LIN {X 0,Y 573.004,Z 629.89,A -85,B 0,C 180,E1 -2246.484,E2 -2246.484} C_VEL
LIN {X 0,Y 572.937,Z 632.192,A -85,B 0,C 180,E1 -2247.891,E2 -2247.891} C_VEL
LIN {X 0,Y 572.938,Z 633.349,A -85,B 0,C 180,E1 -2249.297,E2 -2249.297} C_VEL
LIN {X 0,Y 572.938,Z 633.349,A -85,B 0,C 180,E1 -2250.703,E2 -2250.703} C_VEL
LIN {X 0,Y 572.937,Z 632.19,A -85,B 0,C 180,E1 -2252.109,E2 -2252.109} C_VEL
LIN {X 0,Y 573.004,Z 629.886,A -85,B 0,C 180,E1 -2253.516,E2 -2253.516} C_VEL
LIN {X 0,Y 572.951,Z 626.385,A -85,B 0,C 180,E1 -2254.926,E2 -2254.926} C_VEL
LIN {X 0,Y 573.012,Z 621.608,A -85,B 0,C 180,E1 -2256.338,E2 -2256.338} C_VEL
LIN {X 0,Y 573.094,Z 615.422,A -85,B 0,C 180,E1 -2257.753,E2 -2257.753} C_VEL
LIN {X 0,Y 573.136,Z 607.648,A -85,B 0,C 180,E1 -2259.173,E2 -2259.173} C_VEL
LIN {X 0,Y 573.27,Z 599.368,A -85,B 0,C 180,E1 -2260.418,E2 -2260.418} C_VEL
LIN {X 0,Y 573.386,Z 589.391,A -85,B 0,C 180,E1 -2261.668,E2 -2261.668} C_VEL
LIN {X 0,Y 573.568,Z 579.188,A -85,B 0,C 180,E1 -2262.742,E2 -2262.742} C_VEL
LIN {X 0,Y 573.705,Z 567.019,A -85,B 0,C 180,E1 -2263.82,E2 -2263.82} C_VEL
LIN {X 0,Y 573.963,Z 553.905,A -85,B 0,C 180,E1 -2264.781,E2 -2264.781} C_VEL
LIN {X 0,Y 574.144,Z 539.872,A -85,B 0,C 180,E1 -2265.622,E2 -2265.622} C_VEL
LIN {X 0,Y 574.34,Z 525.8,A -85,B 0,C 180,E1 -2266.301,E2 -2266.301} C_VEL
LIN {X 0,Y 574.564,Z 511.306,A -85,B 0,C 180,E1 -2266.842,E2 -2266.842} C_VEL
LIN {X 0,Y 574.707,Z 496.013,A -85,B 0,C 180,E1 -2267.261,E2 -2267.261} C_VEL
LIN {X 0,Y 574.798,Z 480.641,A -85,B 0,C 180,E1 -2267.532,E2 -2267.532} C_VEL
LIN {X 0,Y 575.183,Z 328.245,A -85,B 0,C 180,E1 -2269.486,E2 -2269.486} C_VEL
LIN {X 0,Y 574.002,Z 321.806,A -85,B 0,C 180,E1 -2269.623,E2 -2269.623} C_VEL
LIN {X 0,Y 574.351,Z 296.393,A -85,B 0,C 180,E1 -2272.671,E2 -2272.671} C_VEL
LIN {X 0,Y 574.622,Z 274.45,A -85,B 0,C 180,E1 -2275.345,E2 -2275.345} C_VEL
LIN {X 0,Y 573.935,Z 269.691,A -85,B 0,C 180,E1 -2275.961,E2 -2275.961} C_VEL
LIN {X 0,Y 573.238,Z 266.709,A -85,B 0,C 180,E1 -2276.376,E2 -2276.376} C_VEL
LIN {X 0,Y 573.259,Z 266.699,A -85,B 0,C 180,E1 -2279.366,E2 -2279.366} C_VEL
LIN {X 0,Y 573.246,Z 266.708,A -85,B 0,C 180,E1 -2282.227,E2 -2282.227} C_VEL
LIN {X 0,Y 573.219,Z 266.705,A -85,B 0,C 180,E1 -2284.769,E2 -2284.769} C_VEL
LIN {X 0,Y 573.22,Z 266.708,A -85,B 0,C 180,E1 -2287.808,E2 -2287.808} C_VEL
LIN {X 0,Y 573.244,Z 266.702,A -85,B 0,C 180,E1 -2290.524,E2 -2290.524} C_VEL
LIN {X 0,Y 573.196,Z 266.705,A -85,B 0,C 180,E1 -2293.362,E2 -2293.362} C_VEL
LIN {X 0,Y 573.203,Z 266.709,A -85,B 0,C 180,E1 -2296.335,E2 -2296.335} C_VEL
LIN {X 0,Y 573.201,Z 266.707,A -85,B 0,C 180,E1 -2298.54,E2 -2298.54} C_VEL
LIN {X 0,Y 573.227,Z 266.701,A -85,B 0,C 180,E1 -2301.297,E2 -2301.297} C_VEL
LIN {X 0,Y 573.181,Z 266.715,A -85,B 0,C 180,E1 -2304.022,E2 -2304.022} C_VEL
LIN {X 0,Y 573.225,Z 266.702,A -85,B 0,C 180,E1 -2306.514,E2 -2306.514} C_VEL
LIN {X 0,Y 573.216,Z 266.703,A -85,B 0,C 180,E1 -2309.119,E2 -2309.119} C_VEL
LIN {X 0,Y 573.215,Z 266.71,A -85,B 0,C 180,E1 -2311.976,E2 -2311.976} C_VEL
LIN {X 0,Y 573.2,Z 266.705,A -85,B 0,C 180,E1 -2314.587,E2 -2314.587} C_VEL
LIN {X 0,Y 573.231,Z 266.7,A -85,B 0,C 180,E1 -2316.9,E2 -2316.9} C_VEL
LIN {X 0,Y 573.241,Z 266.701,A -85,B 0,C 180,E1 -2319.172,E2 -2319.172} C_VEL
LIN {X 0,Y 573.194,Z 266.709,A -85,B 0,C 180,E1 -2321.409,E2 -2321.409} C_VEL
LIN {X 0,Y 573.209,Z 266.704,A -85,B 0,C 180,E1 -2324.35,E2 -2324.35} C_VEL
LIN {X 0,Y 573.201,Z 266.701,A -85,B 0,C 180,E1 -2326.528,E2 -2326.528} C_VEL
LIN {X 0,Y 573.218,Z 266.705,A -85,B 0,C 180,E1 -2329.401,E2 -2329.401} C_VEL
LIN {X 0,Y 573.202,Z 266.705,A -85,B 0,C 180,E1 -2332.248,E2 -2332.248} C_VEL
LIN {X 0,Y 573.283,Z 266.695,A -85,B 0,C 180,E1 -2335.076,E2 -2335.076} C_VEL
LIN {X 0,Y 573.279,Z 266.697,A -85,B 0,C 180,E1 -2337.891,E2 -2337.891} C_VEL
LIN {X 0,Y 573.287,Z 266.696,A -85,B 0,C 180,E1 -2339.999,E2 -2339.999} C_VEL
LIN {X 0,Y 573.266,Z 266.696,A -85,B 0,C 180,E1 -2342.81,E2 -2342.81} C_VEL
LIN {X 0,Y 573.257,Z 266.7,A -85,B 0,C 180,E1 -2345.627,E2 -2345.627} C_VEL
LIN {X 0,Y 573.209,Z 266.701,A -85,B 0,C 180,E1 -2348.459,E2 -2348.459} C_VEL
LIN {X 0,Y 573.26,Z 266.705,A -85,B 0,C 180,E1 -2351.311,E2 -2351.311} C_VEL
LIN {X 0,Y 573.213,Z 266.701,A -85,B 0,C 180,E1 -2354.401,E2 -2354.401} C_VEL
LIN {X 0,Y 573.224,Z 266.703,A -85,B 0,C 180,E1 -2357.111,E2 -2357.111} C_VEL
LIN {X 0,Y 573.214,Z 266.702,A -85,B 0,C 180,E1 -2360.076,E2 -2360.076} C_VEL
LIN {X 0,Y 573.204,Z 266.703,A -85,B 0,C 180,E1 -2362.337,E2 -2362.337} C_VEL
LIN {X 0,Y 573.18,Z 266.706,A -85,B 0,C 180,E1 -2364.332,E2 -2364.332} C_VEL
LIN {X 0,Y 572.541,Z 266.791,A -85,B 0,C 180,E1 -2364.919,E2 -2364.919} C_VEL
LIN {X 0,Y 569.711,Z 267.148,A -85,B 0,C 180,E1 -2365.87,E2 -2365.87} C_VEL
LIN {X 0,Y 567.294,Z 267.45,A -85,B 0,C 180,E1 -2366.636,E2 -2366.636} C_VEL
LIN {X 0,Y 566.238,Z 267.577,A -85,B 0,C 180,E1 -2367.227,E2 -2367.227} C_VEL
LIN {X 0,Y 566.143,Z 267.586,A -85,B 0,C 180,E1 -2367.428,E2 -2367.428} C_VEL
LIN {X 0,Y 566.147,Z 267.584,A -85,B 0,C 180,E1 -2369.77,E2 -2369.77} C_VEL
LIN {X 0,Y 566.183,Z 267.579,A -85,B 0,C 180,E1 -2372.428,E2 -2372.428} C_VEL
LIN {X 0,Y 566.151,Z 267.588,A -85,B 0,C 180,E1 -2374.987,E2 -2374.987} C_VEL
LIN {X 0,Y 566.174,Z 267.582,A -85,B 0,C 180,E1 -2377.46,E2 -2377.46} C_VEL
LIN {X 0,Y 566.19,Z 267.577,A -85,B 0,C 180,E1 -2380.198,E2 -2380.198} C_VEL
LIN {X 0,Y 566.176,Z 267.588,A -85,B 0,C 180,E1 -2383.054,E2 -2383.054} C_VEL
LIN {X 0,Y 566.141,Z 267.581,A -85,B 0,C 180,E1 -2386.052,E2 -2386.052} C_VEL
LIN {X 0,Y 566.153,Z 267.59,A -85,B 0,C 180,E1 -2388.859,E2 -2388.859} C_VEL
LIN {X 0,Y 566.189,Z 267.579,A -85,B 0,C 180,E1 -2391.441,E2 -2391.441} C_VEL
LIN {X 0,Y 566.155,Z 267.582,A -85,B 0,C 180,E1 -2394.308,E2 -2394.308} C_VEL
LIN {X 0,Y 566.185,Z 267.588,A -85,B 0,C 180,E1 -2396.896,E2 -2396.896} C_VEL
LIN {X 0,Y 566.158,Z 267.582,A -85,B 0,C 180,E1 -2399.406,E2 -2399.406} C_VEL
LIN {X 0,Y 566.193,Z 267.577,A -85,B 0,C 180,E1 -2401.857,E2 -2401.857} C_VEL
LIN {X 0,Y 566.189,Z 267.579,A -85,B 0,C 180,E1 -2404.25,E2 -2404.25} C_VEL
LIN {X 0,Y 566.152,Z 267.59,A -85,B 0,C 180,E1 -2406.718,E2 -2406.718} C_VEL
LIN {X 0,Y 566.193,Z 267.576,A -85,B 0,C 180,E1 -2409.662,E2 -2409.662} C_VEL
LIN {X 0,Y 566.179,Z 267.588,A -85,B 0,C 180,E1 -2412.668,E2 -2412.668} C_VEL
LIN {X 0,Y 566.208,Z 267.575,A -85,B 0,C 180,E1 -2415.626,E2 -2415.626} C_VEL
LIN {X 0,Y 566.259,Z 267.579,A -85,B 0,C 180,E1 -2418.652,E2 -2418.652} C_VEL
LIN {X 0,Y 566.187,Z 267.578,A -85,B 0,C 180,E1 -2421.434,E2 -2421.434} C_VEL
LIN {X 0,Y 566.242,Z 267.576,A -85,B 0,C 180,E1 -2424.301,E2 -2424.301} C_VEL
LIN {X 0,Y 566.252,Z 267.572,A -85,B 0,C 180,E1 -2427.866,E2 -2427.866} C_VEL
LIN {X 0,Y 566.294,Z 267.574,A -85,B 0,C 180,E1 -2430.711,E2 -2430.711} C_VEL
LIN {X 0,Y 566.167,Z 267.583,A -85,B 0,C 180,E1 -2433.558,E2 -2433.558} C_VEL
LIN {X 0,Y 566.237,Z 267.575,A -85,B 0,C 180,E1 -2435.698,E2 -2435.698} C_VEL
LIN {X 0,Y 566.214,Z 267.629,A -85,B 0,C 180,E1 -2436.562,E2 -2436.562} C_VEL
LIN {X 0,Y 567.18,Z 272.823,A -85,B 0,C 180,E1 -2437.357,E2 -2437.357} C_VEL
LIN {X 0,Y 566.994,Z 288.919,A -85,B 0,C 180,E1 -2439.632,E2 -2439.632} C_VEL
LIN {X 0,Y 566.937,Z 293.131,A -85,B 0,C 180,E1 -2440.197,E2 -2440.197} C_VEL
LIN {X 0,Y 568.464,Z 300.492,A -85,B 0,C 180,E1 -2440.349,E2 -2440.349} C_VEL
LIN {X 0,Y 568.012,Z 456.718,A -85,B 0,C 180,E1 -2442.391,E2 -2442.391} C_VEL
LIN {X 0,Y 567.847,Z 471.71,A -85,B 0,C 180,E1 -2442.712,E2 -2442.712} C_VEL
LIN {X 0,Y 567.619,Z 487.068,A -85,B 0,C 180,E1 -2443.196,E2 -2443.196} C_VEL
LIN {X 0,Y 567.401,Z 501.304,A -85,B 0,C 180,E1 -2443.794,E2 -2443.794} C_VEL
LIN {X 0,Y 567.186,Z 515.574,A -85,B 0,C 180,E1 -2444.555,E2 -2444.555} C_VEL
LIN {X 0,Y 566.934,Z 529.252,A -85,B 0,C 180,E1 -2445.457,E2 -2445.457} C_VEL
LIN {X 0,Y 566.673,Z 542.03,A -85,B 0,C 180,E1 -2446.481,E2 -2446.481} C_VEL
LIN {X 0,Y 566.461,Z 552.788,A -85,B 0,C 180,E1 -2447.509,E2 -2447.509} C_VEL
LIN {X 0,Y 566.31,Z 562.764,A -85,B 0,C 180,E1 -2448.636,E2 -2448.636} C_VEL
LIN {X 0,Y 566.164,Z 572.566,A -85,B 0,C 180,E1 -2449.959,E2 -2449.959} C_VEL
LIN {X 0,Y 566.028,Z 581.205,A -85,B 0,C 180,E1 -2451.379,E2 -2451.379} C_VEL
LIN {X 0,Y 565.992,Z 587.484,A -85,B 0,C 180,E1 -2452.639,E2 -2452.639} C_VEL
LIN {X 0,Y 565.929,Z 593.647,A -85,B 0,C 180,E1 -2454.192,E2 -2454.192} C_VEL
LIN {X 0,Y 565.877,Z 598.273,A -85,B 0,C 180,E1 -2455.764,E2 -2455.764} C_VEL
LIN {X 0,Y 565.824,Z 601.432,A -85,B 0,C 180,E1 -2457.358,E2 -2457.358} C_VEL
LIN {X 0,Y 565.831,Z 603.143,A -85,B 0,C 180,E1 -2458.973,E2 -2458.973} C_VEL
LIN {X 0,Y 565.866,Z 603.382,A -85,B 0,C 180,E1 -2460.61,E2 -2460.61} C_VEL
LIN {X 0,Y 565.841,Z 602.082,A -85,B 0,C 180,E1 -2462.28,E2 -2462.28} C_VEL
LIN {X 0,Y 565.867,Z 599.727,A -85,B 0,C 180,E1 -2463.685,E2 -2463.685} C_VEL
LIN {X 0,Y 565.899,Z 595.585,A -85,B 0,C 180,E1 -2465.303,E2 -2465.303} C_VEL
LIN {X 0,Y 565.943,Z 591.112,A -85,B 0,C 180,E1 -2466.588,E2 -2466.588} C_VEL
LIN {X 0,Y 566,Z 585.273,A -85,B 0,C 180,E1 -2467.924,E2 -2467.924} C_VEL
LIN {X 0,Y 566.09,Z 577.948,A -85,B 0,C 180,E1 -2469.283,E2 -2469.283} C_VEL
LIN {X 0,Y 566.222,Z 568.957,A -85,B 0,C 180,E1 -2470.648,E2 -2470.648} C_VEL
LIN {X 0,Y 566.322,Z 559.209,A -85,B 0,C 180,E1 -2471.879,E2 -2471.879} C_VEL
LIN {X 0,Y 566.544,Z 548.415,A -85,B 0,C 180,E1 -2473.02,E2 -2473.02} C_VEL
LIN {X 0,Y 566.795,Z 536.367,A -85,B 0,C 180,E1 -2474.087,E2 -2474.087} C_VEL
LIN {X 0,Y 567.041,Z 523.201,A -85,B 0,C 180,E1 -2475.055,E2 -2475.055} C_VEL
LIN {X 0,Y 567.272,Z 509.632,A -85,B 0,C 180,E1 -2475.873,E2 -2475.873} C_VEL
LIN {X 0,Y 567.52,Z 495.08,A -85,B 0,C 180,E1 -2476.575,E2 -2476.575} C_VEL
LIN {X 0,Y 567.733,Z 479.651,A -85,B 0,C 180,E1 -2477.147,E2 -2477.147} C_VEL
LIN {X 0,Y 567.942,Z 464.183,A -85,B 0,C 180,E1 -2477.557,E2 -2477.557} C_VEL
LIN {X 0,Y 568.026,Z 447.504,A -85,B 0,C 180,E1 -2477.834,E2 -2477.834} C_VEL
LIN {X 0,Y 568.365,Z 299.674,A -85,B 0,C 180,E1 -2479.755,E2 -2479.755} C_VEL
LIN {X 0,Y 566.896,Z 292.8,A -85,B 0,C 180,E1 -2479.917,E2 -2479.917} C_VEL
LIN {X 0,Y 567.195,Z 273.626,A -85,B 0,C 180,E1 -2482.619,E2 -2482.619} C_VEL
LIN {X 0,Y 566.221,Z 267.583,A -85,B 0,C 180,E1 -2483.562,E2 -2483.562} C_VEL
LIN {X 0,Y 566.211,Z 267.578,A -85,B 0,C 180,E1 -2486.264,E2 -2486.264} C_VEL
LIN {X 0,Y 566.187,Z 267.581,A -85,B 0,C 180,E1 -2488.922,E2 -2488.922} C_VEL
LIN {X 0,Y 566.182,Z 267.584,A -85,B 0,C 180,E1 -2491.048,E2 -2491.048} C_VEL
LIN {X 0,Y 566.231,Z 267.582,A -85,B 0,C 180,E1 -2493.461,E2 -2493.461} C_VEL
LIN {X 0,Y 566.182,Z 267.583,A -85,B 0,C 180,E1 -2495.82,E2 -2495.82} C_VEL
LIN {X 0,Y 566.201,Z 267.58,A -85,B 0,C 180,E1 -2498.904,E2 -2498.904} C_VEL
LIN {X 0,Y 566.198,Z 267.585,A -85,B 0,C 180,E1 -2501.174,E2 -2501.174} C_VEL
LIN {X 0,Y 566.204,Z 267.583,A -85,B 0,C 180,E1 -2503.414,E2 -2503.414} C_VEL
LIN {X 0,Y 566.186,Z 267.579,A -85,B 0,C 180,E1 -2506.36,E2 -2506.36} C_VEL
LIN {X 0,Y 566.219,Z 267.577,A -85,B 0,C 180,E1 -2508.676,E2 -2508.676} C_VEL
LIN {X 0,Y 566.192,Z 267.582,A -85,B 0,C 180,E1 -2511.435,E2 -2511.435} C_VEL
LIN {X 0,Y 566.246,Z 267.571,A -85,B 0,C 180,E1 -2514.303,E2 -2514.303} C_VEL
LIN {X 0,Y 566.257,Z 267.57,A -85,B 0,C 180,E1 -2517.867,E2 -2517.867} C_VEL
LIN {X 0,Y 566.298,Z 267.571,A -85,B 0,C 180,E1 -2520.712,E2 -2520.712} C_VEL
LIN {X 0,Y 566.264,Z 267.577,A -85,B 0,C 180,E1 -2522.847,E2 -2522.847} C_VEL
LIN {X 0,Y 566.232,Z 267.573,A -85,B 0,C 180,E1 -2525.7,E2 -2525.7} C_VEL
LIN {X 0,Y 566.191,Z 267.577,A -85,B 0,C 180,E1 -2527.849,E2 -2527.849} C_VEL
LIN {X 0,Y 566.225,Z 267.582,A -85,B 0,C 180,E1 -2530.731,E2 -2530.731} C_VEL
LIN {X 0,Y 566.173,Z 267.579,A -85,B 0,C 180,E1 -2533.643,E2 -2533.643} C_VEL
LIN {X 0,Y 566.201,Z 267.585,A -85,B 0,C 180,E1 -2536.589,E2 -2536.589} C_VEL
LIN {X 0,Y 566.19,Z 267.577,A -85,B 0,C 180,E1 -2539.582,E2 -2539.582} C_VEL
LIN {X 0,Y 566.178,Z 267.58,A -85,B 0,C 180,E1 -2541.864,E2 -2541.864} C_VEL
LIN {X 0,Y 566.168,Z 267.582,A -85,B 0,C 180,E1 -2545.022,E2 -2545.022} C_VEL
LIN {X 0,Y 566.153,Z 267.582,A -85,B 0,C 180,E1 -2547.343,E2 -2547.343} C_VEL
LIN {X 0,Y 566.156,Z 267.583,A -85,B 0,C 180,E1 -2549.772,E2 -2549.772} C_VEL
LIN {X 0,Y 566.184,Z 267.587,A -85,B 0,C 180,E1 -2552.429,E2 -2552.429} C_VEL
LIN {X 0,Y 566.15,Z 267.583,A -85,B 0,C 180,E1 -2554.987,E2 -2554.987} C_VEL
LIN {X 0,Y 566.175,Z 267.58,A -85,B 0,C 180,E1 -2557.463,E2 -2557.463} C_VEL
LIN {X 0,Y 566.171,Z 267.59,A -85,B 0,C 180,E1 -2560.203,E2 -2560.203} C_VEL
LIN {X 0,Y 566.172,Z 267.58,A -85,B 0,C 180,E1 -2563.058,E2 -2563.058} C_VEL
LIN {X 0,Y 566.149,Z 267.592,A -85,B 0,C 180,E1 -2566.055,E2 -2566.055} C_VEL
LIN {X 0,Y 566.168,Z 267.581,A -85,B 0,C 180,E1 -2569.219,E2 -2569.219} C_VEL
LIN {X 0,Y 566.171,Z 267.585,A -85,B 0,C 180,E1 -2571.637,E2 -2571.637} C_VEL
LIN {X 0,Y 566.136,Z 267.589,A -85,B 0,C 180,E1 -2574.307,E2 -2574.307} C_VEL
LIN {X 0,Y 566.205,Z 267.577,A -85,B 0,C 180,E1 -2576.898,E2 -2576.898} C_VEL
LIN {X 0,Y 566.174,Z 267.584,A -85,B 0,C 180,E1 -2579.408,E2 -2579.408} C_VEL
LIN {X 0,Y 566.185,Z 267.587,A -85,B 0,C 180,E1 -2581.857,E2 -2581.857} C_VEL
LIN {X 0,Y 566.163,Z 267.606,A -85,B 0,C 180,E1 -2583.425,E2 -2583.425} C_VEL
LIN {X 0,Y 567.69,Z 274.251,A -85,B 0,C 180,E1 -2584.324,E2 -2584.324} C_VEL
LIN {X 0,Y 567.568,Z 291.068,A -85,B 0,C 180,E1 -2586.394,E2 -2586.394} C_VEL
LIN {X 0,Y 567.283,Z 312.004,A -85,B 0,C 180,E1 -2588.945,E2 -2588.945} C_VEL
LIN {X 0,Y 567.116,Z 321.972,A -85,B 0,C 180,E1 -2590.143,E2 -2590.143} C_VEL
LIN {X 0,Y 568.492,Z 329.339,A -85,B 0,C 180,E1 -2590.29,E2 -2590.29} C_VEL
LIN {X 0,Y 567.986,Z 487.947,A -85,B 0,C 180,E1 -2592.364,E2 -2592.364} C_VEL
LIN {X 0,Y 567.854,Z 503.728,A -85,B 0,C 180,E1 -2592.721,E2 -2592.721} C_VEL
LIN {X 0,Y 567.607,Z 519.055,A -85,B 0,C 180,E1 -2593.223,E2 -2593.223} C_VEL
LIN {X 0,Y 567.445,Z 532.788,A -85,B 0,C 180,E1 -2593.82,E2 -2593.82} C_VEL
LIN {X 0,Y 567.151,Z 546.258,A -85,B 0,C 180,E1 -2594.549,E2 -2594.549} C_VEL
LIN {X 0,Y 566.931,Z 558.534,A -85,B 0,C 180,E1 -2595.36,E2 -2595.36} C_VEL
LIN {X 0,Y 566.672,Z 571.298,A -85,B 0,C 180,E1 -2596.371,E2 -2596.371} C_VEL
LIN {X 0,Y 566.491,Z 582.755,A -85,B 0,C 180,E1 -2597.461,E2 -2597.461} C_VEL
LIN {X 0,Y 566.269,Z 593.317,A -85,B 0,C 180,E1 -2598.659,E2 -2598.659} C_VEL
LIN {X 0,Y 566.208,Z 601.86,A -85,B 0,C 180,E1 -2599.813,E2 -2599.813} C_VEL
LIN {X 0,Y 566.057,Z 609.737,A -85,B 0,C 180,E1 -2601.072,E2 -2601.072} C_VEL
LIN {X 0,Y 565.998,Z 617.092,A -85,B 0,C 180,E1 -2602.509,E2 -2602.509} C_VEL
LIN {X 0,Y 565.956,Z 622.924,A -85,B 0,C 180,E1 -2603.941,E2 -2603.941} C_VEL
LIN {X 0,Y 565.866,Z 626.387,A -85,B 0,C 180,E1 -2605.013,E2 -2605.013} C_VEL
LIN {X 0,Y 565.909,Z 629.89,A -85,B 0,C 180,E1 -2606.44,E2 -2606.44} C_VEL
LIN {X 0,Y 565.838,Z 632.192,A -85,B 0,C 180,E1 -2607.865,E2 -2607.865} C_VEL
LIN {X 0,Y 565.838,Z 633.349,A -85,B 0,C 180,E1 -2609.289,E2 -2609.289} C_VEL
LIN {X 0,Y 565.838,Z 633.348,A -85,B 0,C 180,E1 -2610.712,E2 -2610.712} C_VEL
LIN {X 0,Y 565.838,Z 632.189,A -85,B 0,C 180,E1 -2612.136,E2 -2612.136} C_VEL
LIN {X 0,Y 565.909,Z 629.886,A -85,B 0,C 180,E1 -2613.56,E2 -2613.56} C_VEL
LIN {X 0,Y 565.867,Z 626.385,A -85,B 0,C 180,E1 -2614.988,E2 -2614.988} C_VEL
LIN {X 0,Y 565.956,Z 622.924,A -85,B 0,C 180,E1 -2616.059,E2 -2616.059} C_VEL
LIN {X 0,Y 565.998,Z 617.087,A -85,B 0,C 180,E1 -2617.492,E2 -2617.492} C_VEL
LIN {X 0,Y 566.058,Z 609.73,A -85,B 0,C 180,E1 -2618.928,E2 -2618.928} C_VEL
LIN {X 0,Y 566.209,Z 601.855,A -85,B 0,C 180,E1 -2620.188,E2 -2620.188} C_VEL
LIN {X 0,Y 566.31,Z 592.39,A -85,B 0,C 180,E1 -2621.453,E2 -2621.453} C_VEL
LIN {X 0,Y 566.492,Z 582.748,A -85,B 0,C 180,E1 -2622.539,E2 -2622.539} C_VEL
LIN {X 0,Y 566.672,Z 571.295,A -85,B 0,C 180,E1 -2623.629,E2 -2623.629} C_VEL
LIN {X 0,Y 566.929,Z 558.68,A -85,B 0,C 180,E1 -2624.63,E2 -2624.63} C_VEL
LIN {X 0,Y 567.153,Z 546.247,A -85,B 0,C 180,E1 -2625.451,E2 -2625.451} C_VEL
LIN {X 0,Y 567.448,Z 532.77,A -85,B 0,C 180,E1 -2626.181,E2 -2626.181} C_VEL
LIN {X 0,Y 567.612,Z 519.047,A -85,B 0,C 180,E1 -2626.777,E2 -2626.777} C_VEL
LIN {X 0,Y 567.848,Z 503.72,A -85,B 0,C 180,E1 -2627.28,E2 -2627.28} C_VEL
LIN {X 0,Y 567.982,Z 488.303,A -85,B 0,C 180,E1 -2627.63,E2 -2627.63} C_VEL
LIN {X 0,Y 568.496,Z 329.245,A -85,B 0,C 180,E1 -2629.711,E2 -2629.711} C_VEL
LIN {X 0,Y 567.138,Z 321.835,A -85,B 0,C 180,E1 -2629.867,E2 -2629.867} C_VEL
LIN {X 0,Y 567.555,Z 294.798,A -85,B 0,C 180,E1 -2633.151,E2 -2633.151} C_VEL
LIN {X 0,Y 567.801,Z 276.029,A -85,B 0,C 180,E1 -2635.453,E2 -2635.453} C_VEL
LIN {X 0,Y 567.026,Z 271.09,A -85,B 0,C 180,E1 -2636.104,E2 -2636.104} C_VEL
LIN {X 0,Y 566.151,Z 267.591,A -85,B 0,C 180,E1 -2636.598,E2 -2636.598} C_VEL
LIN {X 0,Y 566.181,Z 267.582,A -85,B 0,C 180,E1 -2638.954,E2 -2638.954} C_VEL
LIN {X 0,Y 566.189,Z 267.579,A -85,B 0,C 180,E1 -2641.422,E2 -2641.422} C_VEL
LIN {X 0,Y 566.194,Z 267.585,A -85,B 0,C 180,E1 -2643.957,E2 -2643.957} C_VEL
LIN {X 0,Y 566.173,Z 267.584,A -85,B 0,C 180,E1 -2646.571,E2 -2646.571} C_VEL
LIN {X 0,Y 566.209,Z 267.58,A -85,B 0,C 180,E1 -2649.685,E2 -2649.685} C_VEL
LIN {X 0,Y 566.18,Z 267.578,A -85,B 0,C 180,E1 -2652.914,E2 -2652.914} C_VEL
LIN {X 0,Y 566.154,Z 267.59,A -85,B 0,C 180,E1 -2656.053,E2 -2656.053} C_VEL
LIN {X 0,Y 566.154,Z 267.583,A -85,B 0,C 180,E1 -2658.858,E2 -2658.858} C_VEL
LIN {X 0,Y 566.198,Z 267.578,A -85,B 0,C 180,E1 -2661.442,E2 -2661.442} C_VEL
LIN {X 0,Y 566.136,Z 267.587,A -85,B 0,C 180,E1 -2664.305,E2 -2664.305} C_VEL
LIN {X 0,Y 566.194,Z 267.576,A -85,B 0,C 180,E1 -2666.895,E2 -2666.895} C_VEL
LIN {X 0,Y 566.165,Z 267.583,A -85,B 0,C 180,E1 -2669.406,E2 -2669.406} C_VEL
LIN {X 0,Y 566.183,Z 267.588,A -85,B 0,C 180,E1 -2671.855,E2 -2671.855} C_VEL
LIN {X 0,Y 566.17,Z 267.584,A -85,B 0,C 180,E1 -2674.248,E2 -2674.248} C_VEL
LIN {X 0,Y 566.16,Z 267.581,A -85,B 0,C 180,E1 -2676.719,E2 -2676.719} C_VEL
LIN {X 0,Y 566.196,Z 267.586,A -85,B 0,C 180,E1 -2679.661,E2 -2679.661} C_VEL
LIN {X 0,Y 566.161,Z 267.589,A -85,B 0,C 180,E1 -2681.92,E2 -2681.92} C_VEL
LIN {X 0,Y 566.182,Z 267.578,A -85,B 0,C 180,E1 -2684.889,E2 -2684.889} C_VEL
LIN {X 0,Y 566.171,Z 267.584,A -85,B 0,C 180,E1 -2687.817,E2 -2687.817} C_VEL
LIN {X 0,Y 566.131,Z 267.589,A -85,B 0,C 180,E1 -2689.99,E2 -2689.99} C_VEL
LIN {X 0,Y 566.173,Z 267.582,A -85,B 0,C 180,E1 -2692.151,E2 -2692.151} C_VEL
LIN {X 0,Y 566.255,Z 267.569,A -85,B 0,C 180,E1 -2695.015,E2 -2695.015} C_VEL
LIN {X 0,Y 566.252,Z 267.572,A -85,B 0,C 180,E1 -2697.865,E2 -2697.865} C_VEL
LIN {X 0,Y 566.258,Z 267.572,A -85,B 0,C 180,E1 -2699.999,E2 -2699.999} C_VEL
LIN {X 0,Y 566.236,Z 267.572,A -85,B 0,C 180,E1 -2702.845,E2 -2702.845} C_VEL
LIN {X 0,Y 566.222,Z 267.574,A -85,B 0,C 180,E1 -2705.697,E2 -2705.697} C_VEL
LIN {X 0,Y 566.164,Z 267.578,A -85,B 0,C 180,E1 -2708.565,E2 -2708.565} C_VEL
LIN {X 0,Y 566.226,Z 267.582,A -85,B 0,C 180,E1 -2711.453,E2 -2711.453} C_VEL
LIN {X 0,Y 566.163,Z 267.579,A -85,B 0,C 180,E1 -2714.482,E2 -2714.482} C_VEL
LIN {X 0,Y 566.169,Z 267.584,A -85,B 0,C 180,E1 -2717.331,E2 -2717.331} C_VEL
LIN {X 0,Y 566.184,Z 267.583,A -85,B 0,C 180,E1 -2719.58,E2 -2719.58} C_VEL
LIN {X 0,Y 566.17,Z 267.582,A -85,B 0,C 180,E1 -2721.862,E2 -2721.862} C_VEL
LIN {X 0,Y 566.164,Z 267.585,A -85,B 0,C 180,E1 -2725.02,E2 -2725.02} C_VEL
LIN {X 0,Y 566.143,Z 267.586,A -85,B 0,C 180,E1 -2727.428,E2 -2727.428} C_VEL
LIN {X 0,Y 565.453,Z 267.668,A -85,B 0,C 180,E1 -2728.021,E2 -2728.021} C_VEL
LIN {X 0,Y 562.596,Z 268.027,A -85,B 0,C 180,E1 -2728.985,E2 -2728.985} C_VEL
LIN {X 0,Y 560.204,Z 268.324,A -85,B 0,C 180,E1 -2729.761,E2 -2729.761} C_VEL
LIN {X 0,Y 559.188,Z 268.449,A -85,B 0,C 180,E1 -2730.36,E2 -2730.36} C_VEL
LIN {X 0,Y 559.11,Z 268.46,A -85,B 0,C 180,E1 -2730.563,E2 -2730.563} C_VEL
LIN {X 0,Y 559.134,Z 268.459,A -85,B 0,C 180,E1 -2732.715,E2 -2732.715} C_VEL
LIN {X 0,Y 559.101,Z 268.463,A -85,B 0,C 180,E1 -2735.324,E2 -2735.324} C_VEL
LIN {X 0,Y 559.112,Z 268.457,A -85,B 0,C 180,E1 -2738.017,E2 -2738.017} C_VEL
LIN {X 0,Y 559.136,Z 268.461,A -85,B 0,C 180,E1 -2740.812,E2 -2740.812} C_VEL
LIN {X 0,Y 559.118,Z 268.457,A -85,B 0,C 180,E1 -2743.733,E2 -2743.733} C_VEL
LIN {X 0,Y 559.113,Z 268.462,A -85,B 0,C 180,E1 -2746.804,E2 -2746.804} C_VEL
LIN {X 0,Y 559.136,Z 268.463,A -85,B 0,C 180,E1 -2749.187,E2 -2749.187} C_VEL
LIN {X 0,Y 559.112,Z 268.457,A -85,B 0,C 180,E1 -2751.981,E2 -2751.981} C_VEL
LIN {X 0,Y 559.123,Z 268.463,A -85,B 0,C 180,E1 -2754.785,E2 -2754.785} C_VEL
LIN {X 0,Y 559.135,Z 268.459,A -85,B 0,C 180,E1 -2757.364,E2 -2757.364} C_VEL
LIN {X 0,Y 559.125,Z 268.456,A -85,B 0,C 180,E1 -2760.143,E2 -2760.143} C_VEL
LIN {X 0,Y 559.151,Z 268.458,A -85,B 0,C 180,E1 -2763.172,E2 -2763.172} C_VEL
LIN {X 0,Y 559.135,Z 268.457,A -85,B 0,C 180,E1 -2765.494,E2 -2765.494} C_VEL
LIN {X 0,Y 559.151,Z 268.462,A -85,B 0,C 180,E1 -2768.623,E2 -2768.623} C_VEL
LIN {X 0,Y 559.148,Z 268.463,A -85,B 0,C 180,E1 -2770.926,E2 -2770.926} C_VEL
LIN {X 0,Y 559.145,Z 268.454,A -85,B 0,C 180,E1 -2773.947,E2 -2773.947} C_VEL
LIN {X 0,Y 559.149,Z 268.457,A -85,B 0,C 180,E1 -2776.184,E2 -2776.184} C_VEL
LIN {X 0,Y 559.22,Z 268.448,A -85,B 0,C 180,E1 -2779.134,E2 -2779.134} C_VEL
LIN {X 0,Y 559.181,Z 268.452,A -85,B 0,C 180,E1 -2782.053,E2 -2782.053} C_VEL
LIN {X 0,Y 559.236,Z 268.449,A -85,B 0,C 180,E1 -2784.953,E2 -2784.953} C_VEL
LIN {X 0,Y 559.224,Z 268.447,A -85,B 0,C 180,E1 -2787.839,E2 -2787.839} C_VEL
LIN {X 0,Y 559.263,Z 268.451,A -85,B 0,C 180,E1 -2790.72,E2 -2790.72} C_VEL
LIN {X 0,Y 559.229,Z 268.452,A -85,B 0,C 180,E1 -2792.881,E2 -2792.881} C_VEL
LIN {X 0,Y 559.206,Z 268.452,A -85,B 0,C 180,E1 -2795.77,E2 -2795.77} C_VEL
LIN {X 0,Y 559.167,Z 268.531,A -85,B 0,C 180,E1 -2796.359,E2 -2796.359} C_VEL
LIN {X 0,Y 560.336,Z 275.249,A -85,B 0,C 180,E1 -2797.397,E2 -2797.397} C_VEL
LIN {X 0,Y 559.973,Z 292.95,A -85,B 0,C 180,E1 -2799.937,E2 -2799.937} C_VEL
LIN {X 0,Y 561.717,Z 301.086,A -85,B 0,C 180,E1 -2800.11,E2 -2800.11} C_VEL
LIN {X 0,Y 561.232,Z 457.24,A -85,B 0,C 180,E1 -2802.18,E2 -2802.18} C_VEL
LIN {X 0,Y 561.053,Z 472.26,A -85,B 0,C 180,E1 -2802.512,E2 -2802.512} C_VEL
LIN {X 0,Y 560.826,Z 487.052,A -85,B 0,C 180,E1 -2802.985,E2 -2802.985} C_VEL
LIN {X 0,Y 560.56,Z 501.413,A -85,B 0,C 180,E1 -2803.596,E2 -2803.596} C_VEL
LIN {X 0,Y 560.307,Z 515.278,A -85,B 0,C 180,E1 -2804.342,E2 -2804.342} C_VEL
LIN {X 0,Y 560.02,Z 528.256,A -85,B 0,C 180,E1 -2805.199,E2 -2805.199} C_VEL
LIN {X 0,Y 559.735,Z 541.049,A -85,B 0,C 180,E1 -2806.222,E2 -2806.222} C_VEL
LIN {X 0,Y 559.474,Z 553.109,A -85,B 0,C 180,E1 -2807.384,E2 -2807.384} C_VEL
LIN {X 0,Y 559.294,Z 562.821,A -85,B 0,C 180,E1 -2808.498,E2 -2808.498} C_VEL
LIN {X 0,Y 559.109,Z 572.616,A -85,B 0,C 180,E1 -2809.839,E2 -2809.839} C_VEL
LIN {X 0,Y 558.972,Z 580.774,A -85,B 0,C 180,E1 -2811.19,E2 -2811.19} C_VEL
LIN {X 0,Y 558.901,Z 587.518,A -85,B 0,C 180,E1 -2812.552,E2 -2812.552} C_VEL
LIN {X 0,Y 558.851,Z 593.664,A -85,B 0,C 180,E1 -2814.123,E2 -2814.123} C_VEL
LIN {X 0,Y 558.832,Z 597.299,A -85,B 0,C 180,E1 -2815.314,E2 -2815.314} C_VEL
LIN {X 0,Y 558.732,Z 600.82,A -85,B 0,C 180,E1 -2816.924,E2 -2816.924} C_VEL
LIN {X 0,Y 558.72,Z 602.878,A -85,B 0,C 180,E1 -2818.553,E2 -2818.553} C_VEL
LIN {X 0,Y 558.767,Z 603.472,A -85,B 0,C 180,E1 -2820.205,E2 -2820.205} C_VEL
LIN {X 0,Y 558.748,Z 603.093,A -85,B 0,C 180,E1 -2821.21,E2 -2821.21} C_VEL
LIN {X 0,Y 558.745,Z 601.473,A -85,B 0,C 180,E1 -2822.741,E2 -2822.741} C_VEL
LIN {X 0,Y 558.771,Z 599.408,A -85,B 0,C 180,E1 -2823.893,E2 -2823.893} C_VEL
LIN {X 0,Y 558.805,Z 595.656,A -85,B 0,C 180,E1 -2825.346,E2 -2825.346} C_VEL
LIN {X 0,Y 558.866,Z 590.842,A -85,B 0,C 180,E1 -2826.741,E2 -2826.741} C_VEL
LIN {X 0,Y 558.924,Z 585.23,A -85,B 0,C 180,E1 -2828.033,E2 -2828.033} C_VEL
LIN {X 0,Y 559.048,Z 577.898,A -85,B 0,C 180,E1 -2829.408,E2 -2829.408} C_VEL
LIN {X 0,Y 559.195,Z 568.773,A -85,B 0,C 180,E1 -2830.807,E2 -2830.807} C_VEL
LIN {X 0,Y 559.311,Z 559.799,A -85,B 0,C 180,E1 -2831.96,E2 -2831.96} C_VEL
LIN {X 0,Y 559.561,Z 548.98,A -85,B 0,C 180,E1 -2833.13,E2 -2833.13} C_VEL
LIN {X 0,Y 559.85,Z 536.608,A -85,B 0,C 180,E1 -2834.244,E2 -2834.244} C_VEL
LIN {X 0,Y 560.133,Z 523.59,A -85,B 0,C 180,E1 -2835.217,E2 -2835.217} C_VEL
LIN {X 0,Y 560.41,Z 509.502,A -85,B 0,C 180,E1 -2836.079,E2 -2836.079} C_VEL
LIN {X 0,Y 560.677,Z 495.448,A -85,B 0,C 180,E1 -2836.766,E2 -2836.766} C_VEL
LIN {X 0,Y 560.922,Z 480.168,A -85,B 0,C 180,E1 -2837.344,E2 -2837.344} C_VEL
LIN {X 0,Y 561.153,Z 464.955,A -85,B 0,C 180,E1 -2837.757,E2 -2837.757} C_VEL
LIN {X 0,Y 561.279,Z 449.087,A -85,B 0,C 180,E1 -2838.034,E2 -2838.034} C_VEL
LIN {X 0,Y 561.747,Z 301.083,A -85,B 0,C 180,E1 -2839.979,E2 -2839.979} C_VEL
LIN {X 0,Y 559.998,Z 292.856,A -85,B 0,C 180,E1 -2840.165,E2 -2840.165} C_VEL
LIN {X 0,Y 560.324,Z 274.625,A -85,B 0,C 180,E1 -2842.791,E2 -2842.791} C_VEL
LIN {X 0,Y 559.178,Z 268.461,A -85,B 0,C 180,E1 -2843.771,E2 -2843.771} C_VEL
LIN {X 0,Y 559.16,Z 268.456,A -85,B 0,C 180,E1 -2846.427,E2 -2846.427} C_VEL
LIN {X 0,Y 559.151,Z 268.459,A -85,B 0,C 180,E1 -2848.982,E2 -2848.982} C_VEL
LIN {X 0,Y 559.155,Z 268.462,A -85,B 0,C 180,E1 -2851.619,E2 -2851.619} C_VEL
LIN {X 0,Y 559.183,Z 268.454,A -85,B 0,C 180,E1 -2853.905,E2 -2853.905} C_VEL
LIN {X 0,Y 559.14,Z 268.458,A -85,B 0,C 180,E1 -2856.568,E2 -2856.568} C_VEL
LIN {X 0,Y 559.171,Z 268.461,A -85,B 0,C 180,E1 -2859.397,E2 -2859.397} C_VEL
LIN {X 0,Y 559.141,Z 268.46,A -85,B 0,C 180,E1 -2861.687,E2 -2861.687} C_VEL
LIN {X 0,Y 559.155,Z 268.456,A -85,B 0,C 180,E1 -2863.949,E2 -2863.949} C_VEL
LIN {X 0,Y 559.16,Z 268.454,A -85,B 0,C 180,E1 -2866.185,E2 -2866.185} C_VEL
LIN {X 0,Y 559.179,Z 268.46,A -85,B 0,C 180,E1 -2869.135,E2 -2869.135} C_VEL
LIN {X 0,Y 559.186,Z 268.45,A -85,B 0,C 180,E1 -2872.055,E2 -2872.055} C_VEL
LIN {X 0,Y 559.239,Z 268.452,A -85,B 0,C 180,E1 -2874.954,E2 -2874.954} C_VEL
LIN {X 0,Y 559.229,Z 268.445,A -85,B 0,C 180,E1 -2877.841,E2 -2877.841} C_VEL
LIN {X 0,Y 559.267,Z 268.447,A -85,B 0,C 180,E1 -2880.721,E2 -2880.721} C_VEL
LIN {X 0,Y 559.229,Z 268.454,A -85,B 0,C 180,E1 -2882.883,E2 -2882.883} C_VEL
LIN {X 0,Y 559.202,Z 268.448,A -85,B 0,C 180,E1 -2885.772,E2 -2885.772} C_VEL
LIN {X 0,Y 559.156,Z 268.461,A -85,B 0,C 180,E1 -2888.676,E2 -2888.676} C_VEL
LIN {X 0,Y 559.19,Z 268.449,A -85,B 0,C 180,E1 -2891.602,E2 -2891.602} C_VEL
LIN {X 0,Y 559.19,Z 268.457,A -85,B 0,C 180,E1 -2894.597,E2 -2894.597} C_VEL
LIN {X 0,Y 559.129,Z 268.457,A -85,B 0,C 180,E1 -2897.559,E2 -2897.559} C_VEL
LIN {X 0,Y 559.154,Z 268.455,A -85,B 0,C 180,E1 -2899.839,E2 -2899.839} C_VEL
LIN {X 0,Y 559.127,Z 268.462,A -85,B 0,C 180,E1 -2902.154,E2 -2902.154} C_VEL
LIN {X 0,Y 559.128,Z 268.458,A -85,B 0,C 180,E1 -2905.179,E2 -2905.179} C_VEL
LIN {X 0,Y 559.124,Z 268.467,A -85,B 0,C 180,E1 -2908.375,E2 -2908.375} C_VEL
LIN {X 0,Y 559.114,Z 268.458,A -85,B 0,C 180,E1 -2911.27,E2 -2911.27} C_VEL
LIN {X 0,Y 559.142,Z 268.46,A -85,B 0,C 180,E1 -2913.948,E2 -2913.948} C_VEL
LIN {X 0,Y 559.103,Z 268.46,A -85,B 0,C 180,E1 -2917.112,E2 -2917.112} C_VEL
LIN {X 0,Y 559.144,Z 268.459,A -85,B 0,C 180,E1 -2919.869,E2 -2919.869} C_VEL
LIN {X 0,Y 559.134,Z 268.458,A -85,B 0,C 180,E1 -2922.747,E2 -2922.747} C_VEL
LIN {X 0,Y 559.116,Z 268.464,A -85,B 0,C 180,E1 -2925.765,E2 -2925.765} C_VEL
LIN {X 0,Y 559.111,Z 268.467,A -85,B 0,C 180,E1 -2928.227,E2 -2928.227} C_VEL
LIN {X 0,Y 559.164,Z 268.454,A -85,B 0,C 180,E1 -2931.194,E2 -2931.194} C_VEL
LIN {X 0,Y 559.11,Z 268.466,A -85,B 0,C 180,E1 -2933.788,E2 -2933.788} C_VEL
LIN {X 0,Y 559.156,Z 268.457,A -85,B 0,C 180,E1 -2936.426,E2 -2936.426} C_VEL
LIN {X 0,Y 559.149,Z 268.456,A -85,B 0,C 180,E1 -2938.981,E2 -2938.981} C_VEL
LIN {X 0,Y 559.132,Z 268.467,A -85,B 0,C 180,E1 -2941.626,E2 -2941.626} C_VEL
LIN {X 0,Y 559.137,Z 268.558,A -85,B 0,C 180,E1 -2943.212,E2 -2943.212} C_VEL
LIN {X 0,Y 560.89,Z 276.299,A -85,B 0,C 180,E1 -2944.274,E2 -2944.274} C_VEL
LIN {X 0,Y 560.675,Z 294.604,A -85,B 0,C 180,E1 -2946.549,E2 -2946.549} C_VEL
LIN {X 0,Y 560.292,Z 316.686,A -85,B 0,C 180,E1 -2949.247,E2 -2949.247} C_VEL
LIN {X 0,Y 560.268,Z 322.109,A -85,B 0,C 180,E1 -2949.892,E2 -2949.892} C_VEL
LIN {X 0,Y 561.819,Z 330.83,A -85,B 0,C 180,E1 -2950.066,E2 -2950.066} C_VEL
LIN {X 0,Y 561.233,Z 488.035,A -85,B 0,C 180,E1 -2952.146,E2 -2952.146} C_VEL
LIN {X 0,Y 561.081,Z 503.726,A -85,B 0,C 180,E1 -2952.506,E2 -2952.506} C_VEL
LIN {X 0,Y 560.793,Z 519.052,A -85,B 0,C 180,E1 -2953.013,E2 -2953.013} C_VEL
LIN {X 0,Y 560.606,Z 532.791,A -85,B 0,C 180,E1 -2953.617,E2 -2953.617} C_VEL
LIN {X 0,Y 560.287,Z 546.261,A -85,B 0,C 180,E1 -2954.355,E2 -2954.355} C_VEL
LIN {X 0,Y 559.997,Z 559.314,A -85,B 0,C 180,E1 -2955.231,E2 -2955.231} C_VEL
LIN {X 0,Y 559.722,Z 571.3,A -85,B 0,C 180,E1 -2956.199,E2 -2956.199} C_VEL
LIN {X 0,Y 559.516,Z 582.755,A -85,B 0,C 180,E1 -2957.302,E2 -2957.302} C_VEL
LIN {X 0,Y 559.304,Z 592.394,A -85,B 0,C 180,E1 -2958.402,E2 -2958.402} C_VEL
LIN {X 0,Y 559.168,Z 601.859,A -85,B 0,C 180,E1 -2959.683,E2 -2959.683} C_VEL
LIN {X 0,Y 559.003,Z 609.738,A -85,B 0,C 180,E1 -2960.959,E2 -2960.959} C_VEL
LIN {X 0,Y 558.921,Z 617.092,A -85,B 0,C 180,E1 -2962.414,E2 -2962.414} C_VEL
LIN {X 0,Y 558.839,Z 622.31,A -85,B 0,C 180,E1 -2963.685,E2 -2963.685} C_VEL
LIN {X 0,Y 558.787,Z 626.387,A -85,B 0,C 180,E1 -2964.95,E2 -2964.95} C_VEL
LIN {X 0,Y 558.818,Z 629.89,A -85,B 0,C 180,E1 -2966.395,E2 -2966.395} C_VEL
LIN {X 0,Y 558.744,Z 632.191,A -85,B 0,C 180,E1 -2967.838,E2 -2967.838} C_VEL
LIN {X 0,Y 558.739,Z 633.349,A -85,B 0,C 180,E1 -2969.28,E2 -2969.28} C_VEL
LIN {X 0,Y 558.739,Z 633.348,A -85,B 0,C 180,E1 -2970.721,E2 -2970.721} C_VEL
LIN {X 0,Y 558.744,Z 632.188,A -85,B 0,C 180,E1 -2972.163,E2 -2972.163} C_VEL
LIN {X 0,Y 558.818,Z 629.885,A -85,B 0,C 180,E1 -2973.606,E2 -2973.606} C_VEL
LIN {X 0,Y 558.787,Z 626.386,A -85,B 0,C 180,E1 -2975.051,E2 -2975.051} C_VEL
LIN {X 0,Y 558.844,Z 621.608,A -85,B 0,C 180,E1 -2976.499,E2 -2976.499} C_VEL
LIN {X 0,Y 558.951,Z 615.421,A -85,B 0,C 180,E1 -2977.95,E2 -2977.95} C_VEL
LIN {X 0,Y 559.005,Z 607.645,A -85,B 0,C 180,E1 -2979.407,E2 -2979.407} C_VEL
LIN {X 0,Y 559.217,Z 599.367,A -85,B 0,C 180,E1 -2980.683,E2 -2980.683} C_VEL
LIN {X 0,Y 559.363,Z 589.391,A -85,B 0,C 180,E1 -2981.965,E2 -2981.965} C_VEL
LIN {X 0,Y 559.597,Z 579.186,A -85,B 0,C 180,E1 -2983.065,E2 -2983.065} C_VEL
LIN {X 0,Y 559.825,Z 567.019,A -85,B 0,C 180,E1 -2984.17,E2 -2984.17} C_VEL
LIN {X 0,Y 560.122,Z 554.689,A -85,B 0,C 180,E1 -2985.1,E2 -2985.1} C_VEL
LIN {X 0,Y 560.361,Z 541.51,A -85,B 0,C 180,E1 -2985.923,E2 -2985.923} C_VEL
LIN {X 0,Y 560.668,Z 526.827,A -85,B 0,C 180,E1 -2986.663,E2 -2986.663} C_VEL
LIN {X 0,Y 560.925,Z 512.616,A -85,B 0,C 180,E1 -2987.218,E2 -2987.218} C_VEL
LIN {X 0,Y 561.144,Z 498.151,A -85,B 0,C 180,E1 -2987.637,E2 -2987.637} C_VEL
LIN {X 0,Y 561.236,Z 483.647,A -85,B 0,C 180,E1 -2987.923,E2 -2987.923} C_VEL
LIN {X 0,Y 561.84,Z 330.185,A -85,B 0,C 180,E1 -2989.942,E2 -2989.942} C_VEL
LIN {X 0,Y 560.243,Z 321.909,A -85,B 0,C 180,E1 -2990.113,E2 -2990.113} C_VEL
LIN {X 0,Y 560.681,Z 296.2,A -85,B 0,C 180,E1 -2993.256,E2 -2993.256} C_VEL
LIN {X 0,Y 560.892,Z 276.349,A -85,B 0,C 180,E1 -2995.726,E2 -2995.726} C_VEL
LIN {X 0,Y 559.131,Z 268.464,A -85,B 0,C 180,E1 -2996.836,E2 -2996.836} C_VEL
LIN {X 0,Y 559.146,Z 268.462,A -85,B 0,C 180,E1 -2999.856,E2 -2999.856} C_VEL
LIN {X 0,Y 559.15,Z 268.458,A -85,B 0,C 180,E1 -3002.715,E2 -3002.715} C_VEL
LIN {X 0,Y 559.115,Z 268.461,A -85,B 0,C 180,E1 -3005.324,E2 -3005.324} C_VEL
LIN {X 0,Y 559.124,Z 268.467,A -85,B 0,C 180,E1 -3008.018,E2 -3008.018} C_VEL
LIN {X 0,Y 559.157,Z 268.462,A -85,B 0,C 180,E1 -3009.941,E2 -3009.941} C_VEL
LIN {X 0,Y 559.138,Z 268.456,A -85,B 0,C 180,E1 -3012.745,E2 -3012.745} C_VEL
LIN {X 0,Y 559.121,Z 268.464,A -85,B 0,C 180,E1 -3015.763,E2 -3015.763} C_VEL
LIN {X 0,Y 559.121,Z 268.465,A -85,B 0,C 180,E1 -3018.225,E2 -3018.225} C_VEL
LIN {X 0,Y 559.165,Z 268.452,A -85,B 0,C 180,E1 -3021.192,E2 -3021.192} C_VEL
LIN {X 0,Y 559.11,Z 268.468,A -85,B 0,C 180,E1 -3023.786,E2 -3023.786} C_VEL
LIN {X 0,Y 559.142,Z 268.457,A -85,B 0,C 180,E1 -3026.423,E2 -3026.423} C_VEL
LIN {X 0,Y 559.145,Z 268.455,A -85,B 0,C 180,E1 -3028.979,E2 -3028.979} C_VEL
LIN {X 0,Y 559.129,Z 268.463,A -85,B 0,C 180,E1 -3031.625,E2 -3031.625} C_VEL
LIN {X 0,Y 559.133,Z 268.457,A -85,B 0,C 180,E1 -3034.821,E2 -3034.821} C_VEL
LIN {X 0,Y 559.132,Z 268.467,A -85,B 0,C 180,E1 -3037.846,E2 -3037.846} C_VEL
LIN {X 0,Y 559.187,Z 268.45,A -85,B 0,C 180,E1 -3040.493,E2 -3040.493} C_VEL
LIN {X 0,Y 559.136,Z 268.459,A -85,B 0,C 180,E1 -3043.195,E2 -3043.195} C_VEL
LIN {X 0,Y 559.148,Z 268.453,A -85,B 0,C 180,E1 -3046.183,E2 -3046.183} C_VEL
LIN {X 0,Y 559.149,Z 268.453,A -85,B 0,C 180,E1 -3049.132,E2 -3049.132} C_VEL
LIN {X 0,Y 559.128,Z 268.461,A -85,B 0,C 180,E1 -3052.051,E2 -3052.051} C_VEL
LIN {X 0,Y 559.229,Z 268.444,A -85,B 0,C 180,E1 -3054.952,E2 -3054.952} C_VEL
LIN {X 0,Y 559.225,Z 268.448,A -85,B 0,C 180,E1 -3057.838,E2 -3057.838} C_VEL
LIN {X 0,Y 559.228,Z 268.447,A -85,B 0,C 180,E1 -3059.999,E2 -3059.999} C_VEL
LIN {X 0,Y 559.205,Z 268.449,A -85,B 0,C 180,E1 -3062.88,E2 -3062.88} C_VEL
LIN {X 0,Y 559.189,Z 268.448,A -85,B 0,C 180,E1 -3065.769,E2 -3065.769} C_VEL
LIN {X 0,Y 559.131,Z 268.454,A -85,B 0,C 180,E1 -3068.674,E2 -3068.674} C_VEL
LIN {X 0,Y 559.183,Z 268.457,A -85,B 0,C 180,E1 -3071.599,E2 -3071.599} C_VEL
LIN {X 0,Y 559.14,Z 268.454,A -85,B 0,C 180,E1 -3074.575,E2 -3074.575} C_VEL
LIN {X 0,Y 559.114,Z 268.461,A -85,B 0,C 180,E1 -3077.557,E2 -3077.557} C_VEL
LIN {X 0,Y 559.147,Z 268.456,A -85,B 0,C 180,E1 -3079.837,E2 -3079.837} C_VEL
LIN {X 0,Y 559.116,Z 268.459,A -85,B 0,C 180,E1 -3082.152,E2 -3082.152} C_VEL
LIN {X 0,Y 559.124,Z 268.465,A -85,B 0,C 180,E1 -3085.177,E2 -3085.177} C_VEL
LIN {X 0,Y 559.092,Z 268.46,A -85,B 0,C 180,E1 -3087.715,E2 -3087.715} C_VEL
LIN {X 0,Y 559.11,Z 268.46,A -85,B 0,C 180,E1 -3090.563,E2 -3090.563} C_VEL
LIN {X 0,Y 558.454,Z 268.55,A -85,B 0,C 180,E1 -3091.164,E2 -3091.164} C_VEL
LIN {X 0,Y 555.597,Z 268.905,A -85,B 0,C 180,E1 -3092.141,E2 -3092.141} C_VEL
LIN {X 0,Y 553.179,Z 269.204,A -85,B 0,C 180,E1 -3092.926,E2 -3092.926} C_VEL
LIN {X 0,Y 552.149,Z 269.33,A -85,B 0,C 180,E1 -3093.533,E2 -3093.533} C_VEL
LIN {X 0,Y 552.069,Z 269.337,A -85,B 0,C 180,E1 -3093.738,E2 -3093.738} C_VEL
LIN {X 0,Y 552.081,Z 269.333,A -85,B 0,C 180,E1 -3096.747,E2 -3096.747} C_VEL
LIN {X 0,Y 552.113,Z 269.334,A -85,B 0,C 180,E1 -3099.526,E2 -3099.526} C_VEL
LIN {X 0,Y 552.091,Z 269.335,A -85,B 0,C 180,E1 -3102.427,E2 -3102.427} C_VEL
LIN {X 0,Y 552.059,Z 269.337,A -85,B 0,C 180,E1 -3105.56,E2 -3105.56} C_VEL
LIN {X 0,Y 552.102,Z 269.337,A -85,B 0,C 180,E1 -3108.678,E2 -3108.678} C_VEL
LIN {X 0,Y 552.097,Z 269.334,A -85,B 0,C 180,E1 -3111.41,E2 -3111.41} C_VEL
LIN {X 0,Y 552.07,Z 269.335,A -85,B 0,C 180,E1 -3114.156,E2 -3114.156} C_VEL
LIN {X 0,Y 552.088,Z 269.343,A -85,B 0,C 180,E1 -3116.813,E2 -3116.813} C_VEL
LIN {X 0,Y 552.082,Z 269.334,A -85,B 0,C 180,E1 -3119.39,E2 -3119.39} C_VEL
LIN {X 0,Y 552.077,Z 269.336,A -85,B 0,C 180,E1 -3121.9,E2 -3121.9} C_VEL
LIN {X 0,Y 552.118,Z 269.336,A -85,B 0,C 180,E1 -3124.653,E2 -3124.653} C_VEL
LIN {X 0,Y 552.072,Z 269.337,A -85,B 0,C 180,E1 -3127.548,E2 -3127.548} C_VEL
LIN {X 0,Y 552.129,Z 269.331,A -85,B 0,C 180,E1 -3130.373,E2 -3130.373} C_VEL
LIN {X 0,Y 552.135,Z 269.333,A -85,B 0,C 180,E1 -3132.977,E2 -3132.977} C_VEL
LIN {X 0,Y 552.114,Z 269.332,A -85,B 0,C 180,E1 -3136.004,E2 -3136.004} C_VEL
LIN {X 0,Y 552.18,Z 269.327,A -85,B 0,C 180,E1 -3138.994,E2 -3138.994} C_VEL
LIN {X 0,Y 552.134,Z 269.329,A -85,B 0,C 180,E1 -3141.951,E2 -3141.951} C_VEL
LIN {X 0,Y 552.21,Z 269.325,A -85,B 0,C 180,E1 -3144.889,E2 -3144.889} C_VEL
LIN {X 0,Y 552.197,Z 269.323,A -85,B 0,C 180,E1 -3147.812,E2 -3147.812} C_VEL
LIN {X 0,Y 552.232,Z 269.327,A -85,B 0,C 180,E1 -3150.729,E2 -3150.729} C_VEL
LIN {X 0,Y 552.194,Z 269.328,A -85,B 0,C 180,E1 -3152.918,E2 -3152.918} C_VEL
LIN {X 0,Y 552.176,Z 269.329,A -85,B 0,C 180,E1 -3155.844,E2 -3155.844} C_VEL
LIN {X 0,Y 552.158,Z 269.519,A -85,B 0,C 180,E1 -3156.165,E2 -3156.165} C_VEL
LIN {X 0,Y 553.468,Z 276.707,A -85,B 0,C 180,E1 -3157.295,E2 -3157.295} C_VEL
LIN {X 0,Y 553.098,Z 293.051,A -85,B 0,C 180,E1 -3159.669,E2 -3159.669} C_VEL
LIN {X 0,Y 555.137,Z 302.772,A -85,B 0,C 180,E1 -3159.886,E2 -3159.886} C_VEL
LIN {X 0,Y 554.466,Z 457.744,A -85,B 0,C 180,E1 -3161.965,E2 -3161.965} C_VEL
LIN {X 0,Y 554.269,Z 473.064,A -85,B 0,C 180,E1 -3162.313,E2 -3162.313} C_VEL
LIN {X 0,Y 553.996,Z 488.519,A -85,B 0,C 180,E1 -3162.826,E2 -3162.826} C_VEL
LIN {X 0,Y 553.703,Z 503.408,A -85,B 0,C 180,E1 -3163.487,E2 -3163.487} C_VEL
LIN {X 0,Y 553.397,Z 516.92,A -85,B 0,C 180,E1 -3164.244,E2 -3164.244} C_VEL
LIN {X 0,Y 553.095,Z 528.891,A -85,B 0,C 180,E1 -3165.057,E2 -3165.057} C_VEL
LIN {X 0,Y 552.803,Z 541.119,A -85,B 0,C 180,E1 -3166.052,E2 -3166.052} C_VEL
LIN {X 0,Y 552.506,Z 553.073,A -85,B 0,C 180,E1 -3167.218,E2 -3167.218} C_VEL
LIN {X 0,Y 552.266,Z 562.884,A -85,B 0,C 180,E1 -3168.358,E2 -3168.358} C_VEL
LIN {X 0,Y 552.095,Z 572.022,A -85,B 0,C 180,E1 -3169.617,E2 -3169.617} C_VEL
LIN {X 0,Y 551.906,Z 579.761,A -85,B 0,C 180,E1 -3170.888,E2 -3170.888} C_VEL
LIN {X 0,Y 551.852,Z 585.766,A -85,B 0,C 180,E1 -3172.066,E2 -3172.066} C_VEL
LIN {X 0,Y 551.784,Z 591.769,A -85,B 0,C 180,E1 -3173.506,E2 -3173.506} C_VEL
LIN {X 0,Y 551.744,Z 596.174,A -85,B 0,C 180,E1 -3174.856,E2 -3174.856} C_VEL
LIN {X 0,Y 551.655,Z 600.054,A -85,B 0,C 180,E1 -3176.48,E2 -3176.48} C_VEL
LIN {X 0,Y 551.657,Z 602.478,A -85,B 0,C 180,E1 -3178.122,E2 -3178.122} C_VEL
LIN {X 0,Y 551.654,Z 603.452,A -85,B 0,C 180,E1 -3179.791,E2 -3179.791} C_VEL
LIN {X 0,Y 551.636,Z 602.981,A -85,B 0,C 180,E1 -3181.399,E2 -3181.399} C_VEL
LIN {X 0,Y 551.662,Z 601.471,A -85,B 0,C 180,E1 -3182.777,E2 -3182.777} C_VEL
LIN {X 0,Y 551.692,Z 599.064,A -85,B 0,C 180,E1 -3184.106,E2 -3184.106} C_VEL
LIN {X 0,Y 551.72,Z 595.725,A -85,B 0,C 180,E1 -3185.391,E2 -3185.391} C_VEL
LIN {X 0,Y 551.796,Z 591.058,A -85,B 0,C 180,E1 -3186.77,E2 -3186.77} C_VEL
LIN {X 0,Y 551.859,Z 584.913,A -85,B 0,C 180,E1 -3188.201,E2 -3188.201} C_VEL
LIN {X 0,Y 551.993,Z 577.843,A -85,B 0,C 180,E1 -3189.537,E2 -3189.537} C_VEL
LIN {X 0,Y 552.161,Z 568.699,A -85,B 0,C 180,E1 -3190.956,E2 -3190.956} C_VEL
LIN {X 0,Y 552.358,Z 558.379,A -85,B 0,C 180,E1 -3192.279,E2 -3192.279} C_VEL
LIN {X 0,Y 552.621,Z 548.219,A -85,B 0,C 180,E1 -3193.372,E2 -3193.372} C_VEL
LIN {X 0,Y 552.908,Z 536.24,A -85,B 0,C 180,E1 -3194.457,E2 -3194.457} C_VEL
LIN {X 0,Y 553.244,Z 523.233,A -85,B 0,C 180,E1 -3195.435,E2 -3195.435} C_VEL
LIN {X 0,Y 553.557,Z 509.901,A -85,B 0,C 180,E1 -3196.26,E2 -3196.26} C_VEL
LIN {X 0,Y 553.842,Z 496.297,A -85,B 0,C 180,E1 -3196.941,E2 -3196.941} C_VEL
LIN {X 0,Y 554.131,Z 481.341,A -85,B 0,C 180,E1 -3197.523,E2 -3197.523} C_VEL
LIN {X 0,Y 554.403,Z 465.653,A -85,B 0,C 180,E1 -3197.963,E2 -3197.963} C_VEL
LIN {X 0,Y 554.526,Z 449.705,A -85,B 0,C 180,E1 -3198.253,E2 -3198.253} C_VEL
LIN {X 0,Y 555.01,Z 301.906,A -85,B 0,C 180,E1 -3200.22,E2 -3200.22} C_VEL
LIN {X 0,Y 553.116,Z 293.045,A -85,B 0,C 180,E1 -3200.427,E2 -3200.427} C_VEL
LIN {X 0,Y 553.454,Z 276.104,A -85,B 0,C 180,E1 -3202.898,E2 -3202.898} C_VEL
LIN {X 0,Y 552.124,Z 269.338,A -85,B 0,C 180,E1 -3203.993,E2 -3203.993} C_VEL
LIN {X 0,Y 552.112,Z 269.335,A -85,B 0,C 180,E1 -3206.816,E2 -3206.816} C_VEL
LIN {X 0,Y 552.098,Z 269.343,A -85,B 0,C 180,E1 -3209.392,E2 -3209.392} C_VEL
LIN {X 0,Y 552.111,Z 269.336,A -85,B 0,C 180,E1 -3211.904,E2 -3211.904} C_VEL
LIN {X 0,Y 552.14,Z 269.33,A -85,B 0,C 180,E1 -3214.65,E2 -3214.65} C_VEL
LIN {X 0,Y 552.081,Z 269.342,A -85,B 0,C 180,E1 -3217.55,E2 -3217.55} C_VEL
LIN {X 0,Y 552.133,Z 269.33,A -85,B 0,C 180,E1 -3220.374,E2 -3220.374} C_VEL
LIN {X 0,Y 552.141,Z 269.335,A -85,B 0,C 180,E1 -3222.978,E2 -3222.978} C_VEL
LIN {X 0,Y 552.122,Z 269.331,A -85,B 0,C 180,E1 -3226.006,E2 -3226.006} C_VEL
LIN {X 0,Y 552.147,Z 269.335,A -85,B 0,C 180,E1 -3228.995,E2 -3228.995} C_VEL
LIN {X 0,Y 552.139,Z 269.328,A -85,B 0,C 180,E1 -3231.953,E2 -3231.953} C_VEL
LIN {X 0,Y 552.214,Z 269.326,A -85,B 0,C 180,E1 -3234.89,E2 -3234.89} C_VEL
LIN {X 0,Y 552.202,Z 269.321,A -85,B 0,C 180,E1 -3237.813,E2 -3237.813} C_VEL
LIN {X 0,Y 552.236,Z 269.323,A -85,B 0,C 180,E1 -3240.73,E2 -3240.73} C_VEL
LIN {X 0,Y 552.194,Z 269.331,A -85,B 0,C 180,E1 -3242.919,E2 -3242.919} C_VEL
LIN {X 0,Y 552.174,Z 269.324,A -85,B 0,C 180,E1 -3245.845,E2 -3245.845} C_VEL
LIN {X 0,Y 552.128,Z 269.338,A -85,B 0,C 180,E1 -3248.787,E2 -3248.787} C_VEL
LIN {X 0,Y 552.147,Z 269.327,A -85,B 0,C 180,E1 -3251.752,E2 -3251.752} C_VEL
LIN {X 0,Y 552.125,Z 269.338,A -85,B 0,C 180,E1 -3254.75,E2 -3254.75} C_VEL
LIN {X 0,Y 552.087,Z 269.334,A -85,B 0,C 180,E1 -3257.79,E2 -3257.79} C_VEL
LIN {X 0,Y 552.115,Z 269.334,A -85,B 0,C 180,E1 -3260.103,E2 -3260.103} C_VEL
LIN {X 0,Y 552.078,Z 269.345,A -85,B 0,C 180,E1 -3262.452,E2 -3262.452} C_VEL
LIN {X 0,Y 552.069,Z 269.337,A -85,B 0,C 180,E1 -3265.334,E2 -3265.334} C_VEL
LIN {X 0,Y 552.066,Z 269.342,A -85,B 0,C 180,E1 -3268.102,E2 -3268.102} C_VEL
LIN {X 0,Y 552.077,Z 269.341,A -85,B 0,C 180,E1 -3270.612,E2 -3270.612} C_VEL
LIN {X 0,Y 552.094,Z 269.334,A -85,B 0,C 180,E1 -3273.188,E2 -3273.188} C_VEL
LIN {X 0,Y 552.058,Z 269.341,A -85,B 0,C 180,E1 -3275.846,E2 -3275.846} C_VEL
LIN {X 0,Y 552.102,Z 269.336,A -85,B 0,C 180,E1 -3278.591,E2 -3278.591} C_VEL
LIN {X 0,Y 552.047,Z 269.34,A -85,B 0,C 180,E1 -3281.453,E2 -3281.453} C_VEL
LIN {X 0,Y 552.068,Z 269.341,A -85,B 0,C 180,E1 -3284.531,E2 -3284.531} C_VEL
LIN {X 0,Y 552.075,Z 269.339,A -85,B 0,C 180,E1 -3287.592,E2 -3287.592} C_VEL
LIN {X 0,Y 552.121,Z 269.334,A -85,B 0,C 180,E1 -3290.474,E2 -3290.474} C_VEL
LIN {X 0,Y 552.064,Z 269.338,A -85,B 0,C 180,E1 -3293.324,E2 -3293.324} C_VEL
LIN {X 0,Y 552.119,Z 269.339,A -85,B 0,C 180,E1 -3295.94,E2 -3295.94} C_VEL
LIN {X 0,Y 552.117,Z 269.333,A -85,B 0,C 180,E1 -3298.542,E2 -3298.542} C_VEL
LIN {X 0,Y 552.094,Z 269.341,A -85,B 0,C 180,E1 -3301.444,E2 -3301.444} C_VEL
LIN {X 0,Y 552.102,Z 269.364,A -85,B 0,C 180,E1 -3302.973,E2 -3302.973} C_VEL
LIN {X 0,Y 554.088,Z 278.412,A -85,B 0,C 180,E1 -3304.232,E2 -3304.232} C_VEL
LIN {X 0,Y 553.778,Z 297.553,A -85,B 0,C 180,E1 -3306.635,E2 -3306.635} C_VEL
LIN {X 0,Y 553.333,Z 321.737,A -85,B 0,C 180,E1 -3309.619,E2 -3309.619} C_VEL
LIN {X 0,Y 555.153,Z 332.093,A -85,B 0,C 180,E1 -3309.835,E2 -3309.835} C_VEL
LIN {X 0,Y 554.469,Z 488.148,A -85,B 0,C 180,E1 -3311.923,E2 -3311.923} C_VEL
LIN {X 0,Y 554.316,Z 503.725,A -85,B 0,C 180,E1 -3312.285,E2 -3312.285} C_VEL
LIN {X 0,Y 553.998,Z 519.05,A -85,B 0,C 180,E1 -3312.799,E2 -3312.799} C_VEL
LIN {X 0,Y 553.773,Z 532.794,A -85,B 0,C 180,E1 -3313.409,E2 -3313.409} C_VEL
LIN {X 0,Y 553.405,Z 546.264,A -85,B 0,C 180,E1 -3314.155,E2 -3314.155} C_VEL
LIN {X 0,Y 553.077,Z 560.157,A -85,B 0,C 180,E1 -3315.104,E2 -3315.104} C_VEL
LIN {X 0,Y 552.76,Z 572.361,A -85,B 0,C 180,E1 -3316.115,E2 -3316.115} C_VEL
LIN {X 0,Y 552.482,Z 584.514,A -85,B 0,C 180,E1 -3317.325,E2 -3317.325} C_VEL
LIN {X 0,Y 552.216,Z 594.49,A -85,B 0,C 180,E1 -3318.514,E2 -3318.514} C_VEL
LIN {X 0,Y 552.124,Z 603.089,A -85,B 0,C 180,E1 -3319.735,E2 -3319.735} C_VEL
LIN {X 0,Y 551.921,Z 610.745,A -85,B 0,C 180,E1 -3321.026,E2 -3321.026} C_VEL
LIN {X 0,Y 551.838,Z 617.092,A -85,B 0,C 180,E1 -3322.316,E2 -3322.316} C_VEL
LIN {X 0,Y 551.745,Z 622.649,A -85,B 0,C 180,E1 -3323.704,E2 -3323.704} C_VEL
LIN {X 0,Y 551.713,Z 626.388,A -85,B 0,C 180,E1 -3324.885,E2 -3324.885} C_VEL
LIN {X 0,Y 551.73,Z 629.889,A -85,B 0,C 180,E1 -3326.349,E2 -3326.349} C_VEL
LIN {X 0,Y 551.654,Z 632.191,A -85,B 0,C 180,E1 -3327.81,E2 -3327.81} C_VEL
LIN {X 0,Y 551.639,Z 633.348,A -85,B 0,C 180,E1 -3329.27,E2 -3329.27} C_VEL
LIN {X 0,Y 551.639,Z 633.348,A -85,B 0,C 180,E1 -3330.73,E2 -3330.73} C_VEL
LIN {X 0,Y 551.654,Z 632.188,A -85,B 0,C 180,E1 -3332.191,E2 -3332.191} C_VEL
LIN {X 0,Y 551.73,Z 629.884,A -85,B 0,C 180,E1 -3333.652,E2 -3333.652} C_VEL
LIN {X 0,Y 551.713,Z 626.386,A -85,B 0,C 180,E1 -3335.116,E2 -3335.116} C_VEL
LIN {X 0,Y 551.781,Z 621.608,A -85,B 0,C 180,E1 -3336.583,E2 -3336.583} C_VEL
LIN {X 0,Y 551.877,Z 615.42,A -85,B 0,C 180,E1 -3338.053,E2 -3338.053} C_VEL
LIN {X 0,Y 551.951,Z 607.644,A -85,B 0,C 180,E1 -3339.528,E2 -3339.528} C_VEL
LIN {X 0,Y 552.184,Z 599.367,A -85,B 0,C 180,E1 -3340.821,E2 -3340.821} C_VEL
LIN {X 0,Y 552.353,Z 589.391,A -85,B 0,C 180,E1 -3342.119,E2 -3342.119} C_VEL
LIN {X 0,Y 552.609,Z 579.185,A -85,B 0,C 180,E1 -3343.234,E2 -3343.234} C_VEL
LIN {X 0,Y 552.889,Z 567.019,A -85,B 0,C 180,E1 -3344.352,E2 -3344.352} C_VEL
LIN {X 0,Y 553.243,Z 554.442,A -85,B 0,C 180,E1 -3345.31,E2 -3345.31} C_VEL
LIN {X 0,Y 553.514,Z 541.507,A -85,B 0,C 180,E1 -3346.126,E2 -3346.126} C_VEL
LIN {X 0,Y 553.866,Z 526.824,A -85,B 0,C 180,E1 -3346.873,E2 -3346.873} C_VEL
LIN {X 0,Y 554.143,Z 512.616,A -85,B 0,C 180,E1 -3347.435,E2 -3347.435} C_VEL
LIN {X 0,Y 554.357,Z 497.515,A -85,B 0,C 180,E1 -3347.877,E2 -3347.877} C_VEL
LIN {X 0,Y 554.522,Z 482.141,A -85,B 0,C 180,E1 -3348.171,E2 -3348.171} C_VEL
LIN {X 0,Y 555.058,Z 330.527,A -85,B 0,C 180,E1 -3350.19,E2 -3350.19} C_VEL
LIN {X 0,Y 553.351,Z 321.714,A -85,B 0,C 180,E1 -3350.385,E2 -3350.385} C_VEL
LIN {X 0,Y 553.846,Z 296.025,A -85,B 0,C 180,E1 -3353.56,E2 -3353.56} C_VEL
LIN {X 0,Y 554.097,Z 278.481,A -85,B 0,C 180,E1 -3355.77,E2 -3355.77} C_VEL
LIN {X 0,Y 552.07,Z 269.342,A -85,B 0,C 180,E1 -3357.071,E2 -3357.071} C_VEL
LIN {X 0,Y 552.115,Z 269.336,A -85,B 0,C 180,E1 -3360.05,E2 -3360.05} C_VEL
LIN {X 0,Y 552.108,Z 269.335,A -85,B 0,C 180,E1 -3362.845,E2 -3362.845} C_VEL
LIN {X 0,Y 552.068,Z 269.344,A -85,B 0,C 180,E1 -3365.844,E2 -3365.844} C_VEL
LIN {X 0,Y 552.111,Z 269.336,A -85,B 0,C 180,E1 -3368.589,E2 -3368.589} C_VEL
LIN {X 0,Y 552.074,Z 269.338,A -85,B 0,C 180,E1 -3371.449,E2 -3371.449} C_VEL
LIN {X 0,Y 552.072,Z 269.339,A -85,B 0,C 180,E1 -3374.529,E2 -3374.529} C_VEL
LIN {X 0,Y 552.106,Z 269.335,A -85,B 0,C 180,E1 -3377.586,E2 -3377.586} C_VEL
LIN {X 0,Y 552.123,Z 269.332,A -85,B 0,C 180,E1 -3380.472,E2 -3380.472} C_VEL
LIN {X 0,Y 552.049,Z 269.342,A -85,B 0,C 180,E1 -3383.324,E2 -3383.324} C_VEL
LIN {X 0,Y 552.093,Z 269.34,A -85,B 0,C 180,E1 -3385.936,E2 -3385.936} C_VEL
LIN {X 0,Y 552.117,Z 269.332,A -85,B 0,C 180,E1 -3388.54,E2 -3388.54} C_VEL
LIN {X 0,Y 552.09,Z 269.338,A -85,B 0,C 180,E1 -3391.443,E2 -3391.443} C_VEL
LIN {X 0,Y 552.068,Z 269.34,A -85,B 0,C 180,E1 -3394.352,E2 -3394.352} C_VEL
LIN {X 0,Y 552.087,Z 269.334,A -85,B 0,C 180,E1 -3396.757,E2 -3396.757} C_VEL
LIN {X 0,Y 552.11,Z 269.334,A -85,B 0,C 180,E1 -3399.119,E2 -3399.119} C_VEL
LIN {X 0,Y 552.075,Z 269.34,A -85,B 0,C 180,E1 -3401.442,E2 -3401.442} C_VEL
LIN {X 0,Y 552.08,Z 269.344,A -85,B 0,C 180,E1 -3403.735,E2 -3403.735} C_VEL
LIN {X 0,Y 552.118,Z 269.33,A -85,B 0,C 180,E1 -3406.003,E2 -3406.003} C_VEL
LIN {X 0,Y 552.117,Z 269.328,A -85,B 0,C 180,E1 -3408.991,E2 -3408.991} C_VEL
LIN {X 0,Y 552.098,Z 269.338,A -85,B 0,C 180,E1 -3411.95,E2 -3411.95} C_VEL
LIN {X 0,Y 552.204,Z 269.319,A -85,B 0,C 180,E1 -3414.888,E2 -3414.888} C_VEL
LIN {X 0,Y 552.198,Z 269.323,A -85,B 0,C 180,E1 -3417.811,E2 -3417.811} C_VEL
LIN {X 0,Y 552.199,Z 269.323,A -85,B 0,C 180,E1 -3419.999,E2 -3419.999} C_VEL
LIN {X 0,Y 552.174,Z 269.325,A -85,B 0,C 180,E1 -3422.917,E2 -3422.917} C_VEL
LIN {X 0,Y 552.157,Z 269.322,A -85,B 0,C 180,E1 -3425.843,E2 -3425.843} C_VEL
LIN {X 0,Y 552.105,Z 269.33,A -85,B 0,C 180,E1 -3428.785,E2 -3428.785} C_VEL
LIN {X 0,Y 552.137,Z 269.332,A -85,B 0,C 180,E1 -3431.75,E2 -3431.75} C_VEL
LIN {X 0,Y 552.107,Z 269.331,A -85,B 0,C 180,E1 -3434.748,E2 -3434.748} C_VEL
LIN {X 0,Y 552.073,Z 269.335,A -85,B 0,C 180,E1 -3437.788,E2 -3437.788} C_VEL
LIN {X 0,Y 552.108,Z 269.331,A -85,B 0,C 180,E1 -3440.1,E2 -3440.1} C_VEL
LIN {X 0,Y 552.068,Z 269.337,A -85,B 0,C 180,E1 -3442.45,E2 -3442.45} C_VEL
LIN {X 0,Y 552.068,Z 269.34,A -85,B 0,C 180,E1 -3445.333,E2 -3445.333} C_VEL
LIN {X 0,Y 552.04,Z 269.336,A -85,B 0,C 180,E1 -3448.1,E2 -3448.1} C_VEL
LIN {X 0,Y 552.076,Z 269.336,A -85,B 0,C 180,E1 -3450.609,E2 -3450.609} C_VEL
LIN {X 0,Y 552.089,Z 269.343,A -85,B 0,C 180,E1 -3453.185,E2 -3453.185} C_VEL
LIN {X 0,Y 552.069,Z 269.337,A -85,B 0,C 180,E1 -3453.738,E2 -3453.738} C_VEL
LIN {X 0,Y 551.426,Z 269.416,A -85,B 0,C 180,E1 -3454.347,E2 -3454.347} C_VEL
LIN {X 0,Y 548.615,Z 269.768,A -85,B 0,C 180,E1 -3455.336,E2 -3455.336} C_VEL
LIN {X 0,Y 546.21,Z 270.066,A -85,B 0,C 180,E1 -3456.131,E2 -3456.131} C_VEL
LIN {X 0,Y 545.147,Z 270.199,A -85,B 0,C 180,E1 -3456.745,E2 -3456.745} C_VEL
LIN {X 0,Y 545.044,Z 270.212,A -85,B 0,C 180,E1 -3456.953,E2 -3456.953} C_VEL
LIN {X 0,Y 545.048,Z 270.211,A -85,B 0,C 180,E1 -3460.142,E2 -3460.142} C_VEL
LIN {X 0,Y 545.028,Z 270.22,A -85,B 0,C 180,E1 -3463.109,E2 -3463.109} C_VEL
LIN {X 0,Y 545.028,Z 270.21,A -85,B 0,C 180,E1 -3466.226,E2 -3466.226} C_VEL
LIN {X 0,Y 545.062,Z 270.217,A -85,B 0,C 180,E1 -3468.884,E2 -3468.884} C_VEL
LIN {X 0,Y 545.06,Z 270.217,A -85,B 0,C 180,E1 -3470.817,E2 -3470.817} C_VEL
LIN {X 0,Y 545.025,Z 270.213,A -85,B 0,C 180,E1 -3473.619,E2 -3473.619} C_VEL
LIN {X 0,Y 545.033,Z 270.215,A -85,B 0,C 180,E1 -3476.326,E2 -3476.326} C_VEL
LIN {X 0,Y 545.047,Z 270.216,A -85,B 0,C 180,E1 -3478.951,E2 -3478.951} C_VEL
LIN {X 0,Y 545.064,Z 270.21,A -85,B 0,C 180,E1 -3481.506,E2 -3481.506} C_VEL
LIN {X 0,Y 545.067,Z 270.212,A -85,B 0,C 180,E1 -3484.493,E2 -3484.493} C_VEL
LIN {X 0,Y 545.017,Z 270.219,A -85,B 0,C 180,E1 -3487.242,E2 -3487.242} C_VEL
LIN {X 0,Y 545.101,Z 270.207,A -85,B 0,C 180,E1 -3490.414,E2 -3490.414} C_VEL
LIN {X 0,Y 545.052,Z 270.21,A -85,B 0,C 180,E1 -3493.521,E2 -3493.521} C_VEL
LIN {X 0,Y 545.074,Z 270.208,A -85,B 0,C 180,E1 -3495.819,E2 -3495.819} C_VEL
LIN {X 0,Y 545.129,Z 270.207,A -85,B 0,C 180,E1 -3498.85,E2 -3498.85} C_VEL
LIN {X 0,Y 545.104,Z 270.205,A -85,B 0,C 180,E1 -3501.847,E2 -3501.847} C_VEL
LIN {X 0,Y 545.186,Z 270.202,A -85,B 0,C 180,E1 -3504.823,E2 -3504.823} C_VEL
LIN {X 0,Y 545.17,Z 270.198,A -85,B 0,C 180,E1 -3507.783,E2 -3507.783} C_VEL
LIN {X 0,Y 545.201,Z 270.203,A -85,B 0,C 180,E1 -3510.738,E2 -3510.738} C_VEL
LIN {X 0,Y 545.159,Z 270.205,A -85,B 0,C 180,E1 -3512.955,E2 -3512.955} C_VEL
LIN {X 0,Y 545.145,Z 270.221,A -85,B 0,C 180,E1 -3515.919,E2 -3515.919} C_VEL
LIN {X 0,Y 546.61,Z 278.263,A -85,B 0,C 180,E1 -3517.201,E2 -3517.201} C_VEL
LIN {X 0,Y 546.247,Z 293.181,A -85,B 0,C 180,E1 -3519.394,E2 -3519.394} C_VEL
LIN {X 0,Y 548.416,Z 303.397,A -85,B 0,C 180,E1 -3519.636,E2 -3519.636} C_VEL
LIN {X 0,Y 547.737,Z 457.474,A -85,B 0,C 180,E1 -3521.729,E2 -3521.729} C_VEL
LIN {X 0,Y 547.546,Z 472.456,A -85,B 0,C 180,E1 -3522.069,E2 -3522.069} C_VEL
LIN {X 0,Y 547.282,Z 485.937,A -85,B 0,C 180,E1 -3522.503,E2 -3522.503} C_VEL
LIN {X 0,Y 546.99,Z 499.728,A -85,B 0,C 180,E1 -3523.088,E2 -3523.088} C_VEL
LIN {X 0,Y 546.613,Z 513.954,A -85,B 0,C 180,E1 -3523.855,E2 -3523.855} C_VEL
LIN {X 0,Y 546.253,Z 526.99,A -85,B 0,C 180,E1 -3524.72,E2 -3524.72} C_VEL
LIN {X 0,Y 545.906,Z 539.076,A -85,B 0,C 180,E1 -3525.685,E2 -3525.685} C_VEL
LIN {X 0,Y 545.565,Z 551.196,A -85,B 0,C 180,E1 -3526.848,E2 -3526.848} C_VEL
LIN {X 0,Y 545.316,Z 561.417,A -85,B 0,C 180,E1 -3528.017,E2 -3528.017} C_VEL
LIN {X 0,Y 545.056,Z 571.441,A -85,B 0,C 180,E1 -3529.391,E2 -3529.391} C_VEL
LIN {X 0,Y 544.845,Z 579.803,A -85,B 0,C 180,E1 -3530.776,E2 -3530.776} C_VEL
LIN {X 0,Y 544.771,Z 585.8,A -85,B 0,C 180,E1 -3531.969,E2 -3531.969} C_VEL
LIN {X 0,Y 544.69,Z 592.352,A -85,B 0,C 180,E1 -3533.576,E2 -3533.576} C_VEL
LIN {X 0,Y 544.64,Z 597.33,A -85,B 0,C 180,E1 -3535.202,E2 -3535.202} C_VEL
LIN {X 0,Y 544.541,Z 600.835,A -85,B 0,C 180,E1 -3536.853,E2 -3536.853} C_VEL
LIN {X 0,Y 544.559,Z 602.883,A -85,B 0,C 180,E1 -3538.522,E2 -3538.522} C_VEL
LIN {X 0,Y 544.576,Z 603.47,A -85,B 0,C 180,E1 -3540.218,E2 -3540.218} C_VEL
LIN {X 0,Y 544.54,Z 602.528,A -85,B 0,C 180,E1 -3541.947,E2 -3541.947} C_VEL
LIN {X 0,Y 544.562,Z 601.218,A -85,B 0,C 180,E1 -3542.982,E2 -3542.982} C_VEL
LIN {X 0,Y 544.602,Z 598.027,A -85,B 0,C 180,E1 -3544.597,E2 -3544.597} C_VEL
LIN {X 0,Y 544.667,Z 594.11,A -85,B 0,C 180,E1 -3545.984,E2 -3545.984} C_VEL
LIN {X 0,Y 544.718,Z 589.24,A -85,B 0,C 180,E1 -3547.328,E2 -3547.328} C_VEL
LIN {X 0,Y 544.801,Z 582.895,A -85,B 0,C 180,E1 -3548.729,E2 -3548.729} C_VEL
LIN {X 0,Y 544.971,Z 574.971,A -85,B 0,C 180,E1 -3550.15,E2 -3550.15} C_VEL
LIN {X 0,Y 545.184,Z 566.865,A -85,B 0,C 180,E1 -3551.358,E2 -3551.358} C_VEL
LIN {X 0,Y 545.387,Z 557.332,A -85,B 0,C 180,E1 -3552.562,E2 -3552.562} C_VEL
LIN {X 0,Y 545.657,Z 546.618,A -85,B 0,C 180,E1 -3553.705,E2 -3553.705} C_VEL
LIN {X 0,Y 546.026,Z 534.971,A -85,B 0,C 180,E1 -3554.748,E2 -3554.748} C_VEL
LIN {X 0,Y 546.368,Z 522.512,A -85,B 0,C 180,E1 -3555.683,E2 -3555.683} C_VEL
LIN {X 0,Y 546.733,Z 509.245,A -85,B 0,C 180,E1 -3556.507,E2 -3556.507} C_VEL
LIN {X 0,Y 547.058,Z 495.727,A -85,B 0,C 180,E1 -3557.185,E2 -3557.185} C_VEL
LIN {X 0,Y 547.376,Z 480.642,A -85,B 0,C 180,E1 -3557.772,E2 -3557.772} C_VEL
LIN {X 0,Y 547.661,Z 464.992,A -85,B 0,C 180,E1 -3558.209,E2 -3558.209} C_VEL
LIN {X 0,Y 547.804,Z 449.415,A -85,B 0,C 180,E1 -3558.487,E2 -3558.487} C_VEL
LIN {X 0,Y 548.387,Z 303.115,A -85,B 0,C 180,E1 -3560.459,E2 -3560.459} C_VEL
LIN {X 0,Y 546.224,Z 293.233,A -85,B 0,C 180,E1 -3560.7,E2 -3560.7} C_VEL
LIN {X 0,Y 546.594,Z 277.801,A -85,B 0,C 180,E1 -3562.977,E2 -3562.977} C_VEL
LIN {X 0,Y 545.081,Z 270.214,A -85,B 0,C 180,E1 -3564.22,E2 -3564.22} C_VEL
LIN {X 0,Y 545.066,Z 270.217,A -85,B 0,C 180,E1 -3567.214,E2 -3567.214} C_VEL
LIN {X 0,Y 545.084,Z 270.214,A -85,B 0,C 180,E1 -3569.814,E2 -3569.814} C_VEL
LIN {X 0,Y 545.085,Z 270.21,A -85,B 0,C 180,E1 -3572.825,E2 -3572.825} C_VEL
LIN {X 0,Y 545.036,Z 270.22,A -85,B 0,C 180,E1 -3575.632,E2 -3575.632} C_VEL
LIN {X 0,Y 545.054,Z 270.214,A -85,B 0,C 180,E1 -3578.838,E2 -3578.838} C_VEL
LIN {X 0,Y 545.07,Z 270.216,A -85,B 0,C 180,E1 -3581.197,E2 -3581.197} C_VEL
LIN {X 0,Y 545.061,Z 270.216,A -85,B 0,C 180,E1 -3583.522,E2 -3583.522} C_VEL
LIN {X 0,Y 545.081,Z 270.209,A -85,B 0,C 180,E1 -3585.821,E2 -3585.821} C_VEL
LIN {X 0,Y 545.102,Z 270.21,A -85,B 0,C 180,E1 -3588.85,E2 -3588.85} C_VEL
LIN {X 0,Y 545.109,Z 270.204,A -85,B 0,C 180,E1 -3591.848,E2 -3591.848} C_VEL
LIN {X 0,Y 545.189,Z 270.199,A -85,B 0,C 180,E1 -3594.824,E2 -3594.824} C_VEL
LIN {X 0,Y 545.175,Z 270.196,A -85,B 0,C 180,E1 -3597.785,E2 -3597.785} C_VEL
LIN {X 0,Y 545.205,Z 270.199,A -85,B 0,C 180,E1 -3600.74,E2 -3600.74} C_VEL
LIN {X 0,Y 545.159,Z 270.206,A -85,B 0,C 180,E1 -3602.957,E2 -3602.957} C_VEL
LIN {X 0,Y 545.125,Z 270.202,A -85,B 0,C 180,E1 -3605.921,E2 -3605.921} C_VEL
LIN {X 0,Y 545.077,Z 270.208,A -85,B 0,C 180,E1 -3608.155,E2 -3608.155} C_VEL
LIN {X 0,Y 545.106,Z 270.207,A -85,B 0,C 180,E1 -3611.152,E2 -3611.152} C_VEL
LIN {X 0,Y 545.079,Z 270.209,A -85,B 0,C 180,E1 -3614.181,E2 -3614.181} C_VEL
LIN {X 0,Y 545.064,Z 270.209,A -85,B 0,C 180,E1 -3617.423,E2 -3617.423} C_VEL
LIN {X 0,Y 545.081,Z 270.214,A -85,B 0,C 180,E1 -3620.374,E2 -3620.374} C_VEL
LIN {X 0,Y 545.063,Z 270.209,A -85,B 0,C 180,E1 -3623.561,E2 -3623.561} C_VEL
LIN {X 0,Y 545.026,Z 270.217,A -85,B 0,C 180,E1 -3626.004,E2 -3626.004} C_VEL
LIN {X 0,Y 545.054,Z 270.214,A -85,B 0,C 180,E1 -3628.744,E2 -3628.744} C_VEL
LIN {X 0,Y 545.035,Z 270.213,A -85,B 0,C 180,E1 -3631.677,E2 -3631.677} C_VEL
LIN {X 0,Y 545.035,Z 270.218,A -85,B 0,C 180,E1 -3634.567,E2 -3634.567} C_VEL
LIN {X 0,Y 545.002,Z 270.217,A -85,B 0,C 180,E1 -3637.307,E2 -3637.307} C_VEL
LIN {X 0,Y 545.027,Z 270.222,A -85,B 0,C 180,E1 -3640.147,E2 -3640.147} C_VEL
LIN {X 0,Y 545.011,Z 270.216,A -85,B 0,C 180,E1 -3643.114,E2 -3643.114} C_VEL
LIN {X 0,Y 545.019,Z 270.223,A -85,B 0,C 180,E1 -3646.23,E2 -3646.23} C_VEL
LIN {X 0,Y 545.013,Z 270.217,A -85,B 0,C 180,E1 -3648.881,E2 -3648.881} C_VEL
LIN {X 0,Y 545.04,Z 270.219,A -85,B 0,C 180,E1 -3651.763,E2 -3651.763} C_VEL
LIN {X 0,Y 545.02,Z 270.218,A -85,B 0,C 180,E1 -3654.532,E2 -3654.532} C_VEL
LIN {X 0,Y 545.063,Z 270.212,A -85,B 0,C 180,E1 -3657.212,E2 -3657.212} C_VEL
LIN {X 0,Y 545.059,Z 270.219,A -85,B 0,C 180,E1 -3659.811,E2 -3659.811} C_VEL
LIN {X 0,Y 545.048,Z 270.235,A -85,B 0,C 180,E1 -3662.736,E2 -3662.736} C_VEL
LIN {X 0,Y 547.23,Z 279.94,A -85,B 0,C 180,E1 -3664.11,E2 -3664.11} C_VEL
LIN {X 0,Y 547.004,Z 294.275,A -85,B 0,C 180,E1 -3665.938,E2 -3665.938} C_VEL
LIN {X 0,Y 546.516,Z 316.292,A -85,B 0,C 180,E1 -3668.699,E2 -3668.699} C_VEL
LIN {X 0,Y 546.431,Z 321.565,A -85,B 0,C 180,E1 -3669.356,E2 -3669.356} C_VEL
LIN {X 0,Y 548.471,Z 332.809,A -85,B 0,C 180,E1 -3669.593,E2 -3669.593} C_VEL
LIN {X 0,Y 547.716,Z 488.371,A -85,B 0,C 180,E1 -3671.701,E2 -3671.701} C_VEL
LIN {X 0,Y 547.526,Z 503.604,A -85,B 0,C 180,E1 -3672.058,E2 -3672.058} C_VEL
LIN {X 0,Y 547.213,Z 518.995,A -85,B 0,C 180,E1 -3672.579,E2 -3672.579} C_VEL
LIN {X 0,Y 546.938,Z 532.797,A -85,B 0,C 180,E1 -3673.195,E2 -3673.195} C_VEL
LIN {X 0,Y 546.529,Z 546.264,A -85,B 0,C 180,E1 -3673.951,E2 -3673.951} C_VEL
LIN {X 0,Y 546.148,Z 560.159,A -85,B 0,C 180,E1 -3674.91,E2 -3674.91} C_VEL
LIN {X 0,Y 545.818,Z 572.362,A -85,B 0,C 180,E1 -3675.935,E2 -3675.935} C_VEL
LIN {X 0,Y 545.511,Z 584.514,A -85,B 0,C 180,E1 -3677.16,E2 -3677.16} C_VEL
LIN {X 0,Y 545.175,Z 595.11,A -85,B 0,C 180,E1 -3678.447,E2 -3678.447} C_VEL
LIN {X 0,Y 545.05,Z 604.299,A -85,B 0,C 180,E1 -3679.788,E2 -3679.788} C_VEL
LIN {X 0,Y 544.845,Z 611.752,A -85,B 0,C 180,E1 -3681.096,E2 -3681.096} C_VEL
LIN {X 0,Y 544.745,Z 618.702,A -85,B 0,C 180,E1 -3682.588,E2 -3682.588} C_VEL
LIN {X 0,Y 544.702,Z 624.164,A -85,B 0,C 180,E1 -3684.076,E2 -3684.076} C_VEL
LIN {X 0,Y 544.605,Z 628.292,A -85,B 0,C 180,E1 -3685.56,E2 -3685.56} C_VEL
LIN {X 0,Y 544.644,Z 631.185,A -85,B 0,C 180,E1 -3687.042,E2 -3687.042} C_VEL
LIN {X 0,Y 544.543,Z 632.91,A -85,B 0,C 180,E1 -3688.521,E2 -3688.521} C_VEL
LIN {X 0,Y 544.538,Z 633.5,A -85,B 0,C 180,E1 -3690,E2 -3690} C_VEL
LIN {X 0,Y 544.544,Z 632.908,A -85,B 0,C 180,E1 -3691.479,E2 -3691.479} C_VEL
LIN {X 0,Y 544.644,Z 631.181,A -85,B 0,C 180,E1 -3692.959,E2 -3692.959} C_VEL
LIN {X 0,Y 544.605,Z 628.288,A -85,B 0,C 180,E1 -3694.441,E2 -3694.441} C_VEL
LIN {X 0,Y 544.702,Z 624.165,A -85,B 0,C 180,E1 -3695.925,E2 -3695.925} C_VEL
LIN {X 0,Y 544.746,Z 618.7,A -85,B 0,C 180,E1 -3697.413,E2 -3697.413} C_VEL
LIN {X 0,Y 544.846,Z 611.744,A -85,B 0,C 180,E1 -3698.905,E2 -3698.905} C_VEL
LIN {X 0,Y 545.074,Z 603.081,A -85,B 0,C 180,E1 -3700.4,E2 -3700.4} C_VEL
LIN {X 0,Y 545.238,Z 593.707,A -85,B 0,C 180,E1 -3701.734,E2 -3701.734} C_VEL
LIN {X 0,Y 545.512,Z 584.507,A -85,B 0,C 180,E1 -3702.84,E2 -3702.84} C_VEL
LIN {X 0,Y 545.792,Z 572.36,A -85,B 0,C 180,E1 -3704.066,E2 -3704.066} C_VEL
LIN {X 0,Y 546.194,Z 559.811,A -85,B 0,C 180,E1 -3705.115,E2 -3705.115} C_VEL
LIN {X 0,Y 546.531,Z 546.251,A -85,B 0,C 180,E1 -3706.05,E2 -3706.05} C_VEL
LIN {X 0,Y 546.945,Z 532.776,A -85,B 0,C 180,E1 -3706.805,E2 -3706.805} C_VEL
LIN {X 0,Y 547.195,Z 518.995,A -85,B 0,C 180,E1 -3707.423,E2 -3707.423} C_VEL
LIN {X 0,Y 547.498,Z 503.613,A -85,B 0,C 180,E1 -3707.943,E2 -3707.943} C_VEL
LIN {X 0,Y 547.722,Z 487.911,A -85,B 0,C 180,E1 -3708.309,E2 -3708.309} C_VEL
LIN {X 0,Y 548.405,Z 331.665,A -85,B 0,C 180,E1 -3710.426,E2 -3710.426} C_VEL
LIN {X 0,Y 546.43,Z 321.54,A -85,B 0,C 180,E1 -3710.655,E2 -3710.655} C_VEL
LIN {X 0,Y 546.963,Z 297.6,A -85,B 0,C 180,E1 -3713.652,E2 -3713.652} C_VEL
LIN {X 0,Y 547.276,Z 280.062,A -85,B 0,C 180,E1 -3715.888,E2 -3715.888} C_VEL
LIN {X 0,Y 545.054,Z 270.216,A -85,B 0,C 180,E1 -3717.298,E2 -3717.298} C_VEL
LIN {X 0,Y 545.059,Z 270.214,A -85,B 0,C 180,E1 -3720.242,E2 -3720.242} C_VEL
LIN {X 0,Y 545.071,Z 270.211,A -85,B 0,C 180,E1 -3723.06,E2 -3723.06} C_VEL
LIN {X 0,Y 545.019,Z 270.22,A -85,B 0,C 180,E1 -3725.67,E2 -3725.67} C_VEL
LIN {X 0,Y 545.045,Z 270.221,A -85,B 0,C 180,E1 -3728.237,E2 -3728.237} C_VEL
LIN {X 0,Y 545.026,Z 270.214,A -85,B 0,C 180,E1 -3731.119,E2 -3731.119} C_VEL
LIN {X 0,Y 545.029,Z 270.223,A -85,B 0,C 180,E1 -3734.131,E2 -3734.131} C_VEL
LIN {X 0,Y 545.021,Z 270.215,A -85,B 0,C 180,E1 -3736.887,E2 -3736.887} C_VEL
LIN {X 0,Y 545.055,Z 270.22,A -85,B 0,C 180,E1 -3739.856,E2 -3739.856} C_VEL
LIN {X 0,Y 545.009,Z 270.218,A -85,B 0,C 180,E1 -3742.693,E2 -3742.693} C_VEL
LIN {X 0,Y 545.05,Z 270.215,A -85,B 0,C 180,E1 -3745.611,E2 -3745.611} C_VEL
LIN {X 0,Y 545.055,Z 270.214,A -85,B 0,C 180,E1 -3748.32,E2 -3748.32} C_VEL
LIN {X 0,Y 545.06,Z 270.212,A -85,B 0,C 180,E1 -3751.256,E2 -3751.256} C_VEL
LIN {X 0,Y 545.03,Z 270.221,A -85,B 0,C 180,E1 -3753.996,E2 -3753.996} C_VEL
LIN {X 0,Y 545.068,Z 270.21,A -85,B 0,C 180,E1 -3756.439,E2 -3756.439} C_VEL
LIN {X 0,Y 545.085,Z 270.215,A -85,B 0,C 180,E1 -3759.627,E2 -3759.627} C_VEL
LIN {X 0,Y 545.043,Z 270.213,A -85,B 0,C 180,E1 -3762.747,E2 -3762.747} C_VEL
LIN {X 0,Y 545.081,Z 270.209,A -85,B 0,C 180,E1 -3765.819,E2 -3765.819} C_VEL
LIN {X 0,Y 545.066,Z 270.205,A -85,B 0,C 180,E1 -3768.847,E2 -3768.847} C_VEL
LIN {X 0,Y 545.056,Z 270.216,A -85,B 0,C 180,E1 -3771.845,E2 -3771.845} C_VEL
LIN {X 0,Y 545.16,Z 270.195,A -85,B 0,C 180,E1 -3774.821,E2 -3774.821} C_VEL
LIN {X 0,Y 545.171,Z 270.199,A -85,B 0,C 180,E1 -3777.782,E2 -3777.782} C_VEL
LIN {X 0,Y 545.169,Z 270.199,A -85,B 0,C 180,E1 -3779.999,E2 -3779.999} C_VEL
LIN {X 0,Y 545.142,Z 270.201,A -85,B 0,C 180,E1 -3782.955,E2 -3782.955} C_VEL
LIN {X 0,Y 545.105,Z 270.199,A -85,B 0,C 180,E1 -3785.919,E2 -3785.919} C_VEL
LIN {X 0,Y 545.05,Z 270.209,A -85,B 0,C 180,E1 -3788.9,E2 -3788.9} C_VEL
LIN {X 0,Y 545.079,Z 270.21,A -85,B 0,C 180,E1 -3791.904,E2 -3791.904} C_VEL
LIN {X 0,Y 545.063,Z 270.21,A -85,B 0,C 180,E1 -3794.943,E2 -3794.943} C_VEL
LIN {X 0,Y 545.039,Z 270.208,A -85,B 0,C 180,E1 -3798.025,E2 -3798.025} C_VEL
LIN {X 0,Y 545.075,Z 270.207,A -85,B 0,C 180,E1 -3800.371,E2 -3800.371} C_VEL
LIN {X 0,Y 545.055,Z 270.214,A -85,B 0,C 180,E1 -3803.559,E2 -3803.559} C_VEL
LIN {X 0,Y 545.028,Z 270.208,A -85,B 0,C 180,E1 -3806.001,E2 -3806.001} C_VEL
LIN {X 0,Y 545.028,Z 270.211,A -85,B 0,C 180,E1 -3808.738,E2 -3808.738} C_VEL
LIN {X 0,Y 545.042,Z 270.215,A -85,B 0,C 180,E1 -3811.678,E2 -3811.678} C_VEL
LIN {X 0,Y 545.03,Z 270.213,A -85,B 0,C 180,E1 -3814.565,E2 -3814.565} C_VEL
LIN {X 0,Y 545.044,Z 270.212,A -85,B 0,C 180,E1 -3816.953,E2 -3816.953} C_VEL
LIN {X 0,Y 544.338,Z 270.302,A -85,B 0,C 180,E1 -3817.57,E2 -3817.57} C_VEL
LIN {X 0,Y 541.481,Z 270.658,A -85,B 0,C 180,E1 -3818.571,E2 -3818.571} C_VEL
LIN {X 0,Y 539.091,Z 270.958,A -85,B 0,C 180,E1 -3819.377,E2 -3819.377} C_VEL
LIN {X 0,Y 538.065,Z 271.081,A -85,B 0,C 180,E1 -3819.999,E2 -3819.999} C_VEL
LIN {X 0,Y 537.98,Z 271.092,A -85,B 0,C 180,E1 -3820.209,E2 -3820.209} C_VEL
LIN {X 0,Y 537.981,Z 271.1,A -85,B 0,C 180,E1 -3822.983,E2 -3822.983} C_VEL
LIN {X 0,Y 537.994,Z 271.086,A -85,B 0,C 180,E1 -3825.927,E2 -3825.927} C_VEL
LIN {X 0,Y 538.03,Z 271.092,A -85,B 0,C 180,E1 -3829.252,E2 -3829.252} C_VEL
LIN {X 0,Y 537.972,Z 271.091,A -85,B 0,C 180,E1 -3832.121,E2 -3832.121} C_VEL
LIN {X 0,Y 537.987,Z 271.098,A -85,B 0,C 180,E1 -3834.915,E2 -3834.915} C_VEL
LIN {X 0,Y 537.998,Z 271.09,A -85,B 0,C 180,E1 -3837.616,E2 -3837.616} C_VEL
LIN {X 0,Y 537.994,Z 271.088,A -85,B 0,C 180,E1 -3840.238,E2 -3840.238} C_VEL
LIN {X 0,Y 538.037,Z 271.093,A -85,B 0,C 180,E1 -3842.795,E2 -3842.795} C_VEL
LIN {X 0,Y 538.003,Z 271.091,A -85,B 0,C 180,E1 -3845.291,E2 -3845.291} C_VEL
LIN {X 0,Y 537.996,Z 271.091,A -85,B 0,C 180,E1 -3848.041,E2 -3848.041} C_VEL
LIN {X 0,Y 538.017,Z 271.095,A -85,B 0,C 180,E1 -3850.939,E2 -3850.939} C_VEL
LIN {X 0,Y 538.003,Z 271.089,A -85,B 0,C 180,E1 -3853.298,E2 -3853.298} C_VEL
LIN {X 0,Y 538.043,Z 271.084,A -85,B 0,C 180,E1 -3855.63,E2 -3855.63} C_VEL
LIN {X 0,Y 538.082,Z 271.087,A -85,B 0,C 180,E1 -3858.702,E2 -3858.702} C_VEL
LIN {X 0,Y 538.062,Z 271.082,A -85,B 0,C 180,E1 -3861.739,E2 -3861.739} C_VEL
LIN {X 0,Y 538.143,Z 271.08,A -85,B 0,C 180,E1 -3864.755,E2 -3864.755} C_VEL
LIN {X 0,Y 538.142,Z 271.074,A -85,B 0,C 180,E1 -3867.754,E2 -3867.754} C_VEL
LIN {X 0,Y 538.17,Z 271.079,A -85,B 0,C 180,E1 -3870.748,E2 -3870.748} C_VEL
LIN {X 0,Y 538.125,Z 271.081,A -85,B 0,C 180,E1 -3872.994,E2 -3872.994} C_VEL
LIN {X 0,Y 538.129,Z 271.26,A -85,B 0,C 180,E1 -3875.715,E2 -3875.715} C_VEL
LIN {X 0,Y 539.752,Z 279.84,A -85,B 0,C 180,E1 -3877.105,E2 -3877.105} C_VEL
LIN {X 0,Y 539.392,Z 293.48,A -85,B 0,C 180,E1 -3879.136,E2 -3879.136} C_VEL
LIN {X 0,Y 541.773,Z 304.418,A -85,B 0,C 180,E1 -3879.387,E2 -3879.387} C_VEL
LIN {X 0,Y 541.006,Z 457.741,A -85,B 0,C 180,E1 -3881.497,E2 -3881.497} C_VEL
LIN {X 0,Y 540.777,Z 472.499,A -85,B 0,C 180,E1 -3881.834,E2 -3881.834} C_VEL
LIN {X 0,Y 540.503,Z 486.184,A -85,B 0,C 180,E1 -3882.281,E2 -3882.281} C_VEL
LIN {X 0,Y 540.185,Z 499.956,A -85,B 0,C 180,E1 -3882.873,E2 -3882.873} C_VEL
LIN {X 0,Y 539.763,Z 514.204,A -85,B 0,C 180,E1 -3883.65,E2 -3883.65} C_VEL
LIN {X 0,Y 539.387,Z 527.199,A -85,B 0,C 180,E1 -3884.525,E2 -3884.525} C_VEL
LIN {X 0,Y 538.987,Z 539.39,A -85,B 0,C 180,E1 -3885.516,E2 -3885.516} C_VEL
LIN {X 0,Y 538.591,Z 551.314,A -85,B 0,C 180,E1 -3886.682,E2 -3886.682} C_VEL
LIN {X 0,Y 538.287,Z 561.722,A -85,B 0,C 180,E1 -3887.898,E2 -3887.898} C_VEL
LIN {X 0,Y 538.023,Z 571.487,A -85,B 0,C 180,E1 -3889.258,E2 -3889.258} C_VEL
LIN {X 0,Y 537.803,Z 579.835,A -85,B 0,C 180,E1 -3890.66,E2 -3890.66} C_VEL
LIN {X 0,Y 537.7,Z 585.881,A -85,B 0,C 180,E1 -3891.88,E2 -3891.88} C_VEL
LIN {X 0,Y 537.614,Z 592.16,A -85,B 0,C 180,E1 -3893.439,E2 -3893.439} C_VEL
LIN {X 0,Y 537.561,Z 596.206,A -85,B 0,C 180,E1 -3894.73,E2 -3894.73} C_VEL
LIN {X 0,Y 537.551,Z 598.339,A -85,B 0,C 180,E1 -3895.568,E2 -3895.568} C_VEL
LIN {X 0,Y 537.436,Z 601.462,A -85,B 0,C 180,E1 -3897.237,E2 -3897.237} C_VEL
LIN {X 0,Y 537.452,Z 603.155,A -85,B 0,C 180,E1 -3898.935,E2 -3898.935} C_VEL
LIN {X 0,Y 537.451,Z 603.377,A -85,B 0,C 180,E1 -3900.662,E2 -3900.662} C_VEL
LIN {X 0,Y 537.439,Z 602.716,A -85,B 0,C 180,E1 -3901.793,E2 -3901.793} C_VEL
LIN {X 0,Y 537.456,Z 600.79,A -85,B 0,C 180,E1 -3903.312,E2 -3903.312} C_VEL
LIN {X 0,Y 537.502,Z 598.294,A -85,B 0,C 180,E1 -3904.542,E2 -3904.542} C_VEL
LIN {X 0,Y 537.573,Z 594.196,A -85,B 0,C 180,E1 -3906.036,E2 -3906.036} C_VEL
LIN {X 0,Y 537.635,Z 588.984,A -85,B 0,C 180,E1 -3907.485,E2 -3907.485} C_VEL
LIN {X 0,Y 537.746,Z 582.855,A -85,B 0,C 180,E1 -3908.852,E2 -3908.852} C_VEL
LIN {X 0,Y 537.94,Z 575.009,A -85,B 0,C 180,E1 -3910.277,E2 -3910.277} C_VEL
LIN {X 0,Y 538.143,Z 566.84,A -85,B 0,C 180,E1 -3911.511,E2 -3911.511} C_VEL
LIN {X 0,Y 538.444,Z 555.939,A -85,B 0,C 180,E1 -3912.896,E2 -3912.896} C_VEL
LIN {X 0,Y 538.804,Z 544.568,A -85,B 0,C 180,E1 -3914.096,E2 -3914.096} C_VEL
LIN {X 0,Y 539.233,Z 532.415,A -85,B 0,C 180,E1 -3915.163,E2 -3915.163} C_VEL
LIN {X 0,Y 539.628,Z 518.972,A -85,B 0,C 180,E1 -3916.14,E2 -3916.14} C_VEL
LIN {X 0,Y 540.048,Z 504.88,A -85,B 0,C 180,E1 -3916.969,E2 -3916.969} C_VEL
LIN {X 0,Y 540.429,Z 490.313,A -85,B 0,C 180,E1 -3917.646,E2 -3917.646} C_VEL
LIN {X 0,Y 540.724,Z 475.812,A -85,B 0,C 180,E1 -3918.16,E2 -3918.16} C_VEL
LIN {X 0,Y 540.996,Z 460.046,A -85,B 0,C 180,E1 -3918.55,E2 -3918.55} C_VEL
LIN {X 0,Y 541.161,Z 430.263,A -85,B 0,C 180,E1 -3918.984,E2 -3918.984} C_VEL
LIN {X 0,Y 541.72,Z 304.129,A -85,B 0,C 180,E1 -3920.711,E2 -3920.711} C_VEL
LIN {X 0,Y 539.419,Z 293.527,A -85,B 0,C 180,E1 -3920.962,E2 -3920.962} C_VEL
LIN {X 0,Y 539.756,Z 280.524,A -85,B 0,C 180,E1 -3922.902,E2 -3922.902} C_VEL
LIN {X 0,Y 538.842,Z 274.727,A -85,B 0,C 180,E1 -3923.833,E2 -3923.833} C_VEL
LIN {X 0,Y 538.032,Z 271.092,A -85,B 0,C 180,E1 -3924.462,E2 -3924.462} C_VEL
LIN {X 0,Y 538.015,Z 271.097,A -85,B 0,C 180,E1 -3927.619,E2 -3927.619} C_VEL
LIN {X 0,Y 538.026,Z 271.089,A -85,B 0,C 180,E1 -3930.241,E2 -3930.241} C_VEL
LIN {X 0,Y 538.055,Z 271.086,A -85,B 0,C 180,E1 -3932.798,E2 -3932.798} C_VEL
LIN {X 0,Y 538.033,Z 271.093,A -85,B 0,C 180,E1 -3935.294,E2 -3935.294} C_VEL
LIN {X 0,Y 537.999,Z 271.091,A -85,B 0,C 180,E1 -3938.043,E2 -3938.043} C_VEL
LIN {X 0,Y 538.026,Z 271.092,A -85,B 0,C 180,E1 -3940.941,E2 -3940.941} C_VEL
LIN {X 0,Y 538.012,Z 271.097,A -85,B 0,C 180,E1 -3943.3,E2 -3943.3} C_VEL
LIN {X 0,Y 538.049,Z 271.087,A -85,B 0,C 180,E1 -3945.632,E2 -3945.632} C_VEL
LIN {X 0,Y 538.062,Z 271.086,A -85,B 0,C 180,E1 -3948.703,E2 -3948.703} C_VEL
LIN {X 0,Y 538.066,Z 271.082,A -85,B 0,C 180,E1 -3951.741,E2 -3951.741} C_VEL
LIN {X 0,Y 538.147,Z 271.076,A -85,B 0,C 180,E1 -3954.756,E2 -3954.756} C_VEL
LIN {X 0,Y 538.147,Z 271.072,A -85,B 0,C 180,E1 -3957.756,E2 -3957.756} C_VEL
LIN {X 0,Y 538.174,Z 271.075,A -85,B 0,C 180,E1 -3960.749,E2 -3960.749} C_VEL
LIN {X 0,Y 538.125,Z 271.082,A -85,B 0,C 180,E1 -3962.996,E2 -3962.996} C_VEL
LIN {X 0,Y 538.081,Z 271.08,A -85,B 0,C 180,E1 -3965.999,E2 -3965.999} C_VEL
LIN {X 0,Y 538.043,Z 271.085,A -85,B 0,C 180,E1 -3968.262,E2 -3968.262} C_VEL
LIN {X 0,Y 538.074,Z 271.08,A -85,B 0,C 180,E1 -3971.6,E2 -3971.6} C_VEL
LIN {X 0,Y 538.048,Z 271.09,A -85,B 0,C 180,E1 -3974.858,E2 -3974.858} C_VEL
LIN {X 0,Y 538.026,Z 271.086,A -85,B 0,C 180,E1 -3977.534,E2 -3977.534} C_VEL
LIN {X 0,Y 538.026,Z 271.095,A -85,B 0,C 180,E1 -3980.653,E2 -3980.653} C_VEL
LIN {X 0,Y 537.997,Z 271.09,A -85,B 0,C 180,E1 -3983.879,E2 -3983.879} C_VEL
LIN {X 0,Y 537.971,Z 271.1,A -85,B 0,C 180,E1 -3986.371,E2 -3986.371} C_VEL
LIN {X 0,Y 538.022,Z 271.088,A -85,B 0,C 180,E1 -3988.934,E2 -3988.934} C_VEL
LIN {X 0,Y 537.989,Z 271.092,A -85,B 0,C 180,E1 -3991.886,E2 -3991.886} C_VEL
LIN {X 0,Y 537.985,Z 271.096,A -85,B 0,C 180,E1 -3994.616,E2 -3994.616} C_VEL
LIN {X 0,Y 537.971,Z 271.096,A -85,B 0,C 180,E1 -3997.88,E2 -3997.88} C_VEL
LIN {X 0,Y 537.98,Z 271.093,A -85,B 0,C 180,E1 -4000.783,E2 -4000.783} C_VEL
LIN {X 0,Y 537.995,Z 271.098,A -85,B 0,C 180,E1 -4004.072,E2 -4004.072} C_VEL
LIN {X 0,Y 537.963,Z 271.095,A -85,B 0,C 180,E1 -4007.02,E2 -4007.02} C_VEL
LIN {X 0,Y 538.001,Z 271.097,A -85,B 0,C 180,E1 -4010.203,E2 -4010.203} C_VEL
LIN {X 0,Y 537.966,Z 271.092,A -85,B 0,C 180,E1 -4013.064,E2 -4013.064} C_VEL
LIN {X 0,Y 538.003,Z 271.096,A -85,B 0,C 180,E1 -4015.827,E2 -4015.827} C_VEL
LIN {X 0,Y 538.006,Z 271.092,A -85,B 0,C 180,E1 -4018.5,E2 -4018.5} C_VEL
LIN {X 0,Y 538.016,Z 271.092,A -85,B 0,C 180,E1 -4021.098,E2 -4021.098} C_VEL
LIN {X 0,Y 538.011,Z 271.104,A -85,B 0,C 180,E1 -4022.492,E2 -4022.492} C_VEL
LIN {X 0,Y 540.417,Z 281.688,A -85,B 0,C 180,E1 -4024.016,E2 -4024.016} C_VEL
LIN {X 0,Y 540.073,Z 298.709,A -85,B 0,C 180,E1 -4026.21,E2 -4026.21} C_VEL
LIN {X 0,Y 539.509,Z 321.334,A -85,B 0,C 180,E1 -4029.079,E2 -4029.079} C_VEL
LIN {X 0,Y 541.82,Z 333.783,A -85,B 0,C 180,E1 -4029.349,E2 -4029.349} C_VEL
LIN {X 0,Y 540.986,Z 487.44,A -85,B 0,C 180,E1 -4031.455,E2 -4031.455} C_VEL
LIN {X 0,Y 540.776,Z 503.262,A -85,B 0,C 180,E1 -4031.827,E2 -4031.827} C_VEL
LIN {X 0,Y 540.41,Z 518.688,A -85,B 0,C 180,E1 -4032.352,E2 -4032.352} C_VEL
LIN {X 0,Y 540.086,Z 532.512,A -85,B 0,C 180,E1 -4032.976,E2 -4032.976} C_VEL
LIN {X 0,Y 539.641,Z 546.058,A -85,B 0,C 180,E1 -4033.74,E2 -4033.74} C_VEL
LIN {X 0,Y 539.308,Z 559.208,A -85,B 0,C 180,E1 -4034.652,E2 -4034.652} C_VEL
LIN {X 0,Y 538.888,Z 571.251,A -85,B 0,C 180,E1 -4035.654,E2 -4035.654} C_VEL
LIN {X 0,Y 538.594,Z 582.752,A -85,B 0,C 180,E1 -4036.8,E2 -4036.8} C_VEL
LIN {X 0,Y 538.283,Z 592.392,A -85,B 0,C 180,E1 -4037.943,E2 -4037.943} C_VEL
LIN {X 0,Y 538.068,Z 601.856,A -85,B 0,C 180,E1 -4039.274,E2 -4039.274} C_VEL
LIN {X 0,Y 537.825,Z 609.737,A -85,B 0,C 180,E1 -4040.6,E2 -4040.6} C_VEL
LIN {X 0,Y 537.7,Z 617.091,A -85,B 0,C 180,E1 -4042.112,E2 -4042.112} C_VEL
LIN {X 0,Y 537.602,Z 622.471,A -85,B 0,C 180,E1 -4043.484,E2 -4043.484} C_VEL
LIN {X 0,Y 537.574,Z 626.387,A -85,B 0,C 180,E1 -4044.75,E2 -4044.75} C_VEL
LIN {X 0,Y 537.561,Z 629.888,A -85,B 0,C 180,E1 -4046.252,E2 -4046.252} C_VEL
LIN {X 0,Y 537.487,Z 632.19,A -85,B 0,C 180,E1 -4047.752,E2 -4047.752} C_VEL
LIN {X 0,Y 537.439,Z 633.348,A -85,B 0,C 180,E1 -4049.251,E2 -4049.251} C_VEL
LIN {X 0,Y 537.439,Z 633.347,A -85,B 0,C 180,E1 -4050.75,E2 -4050.75} C_VEL
LIN {X 0,Y 537.487,Z 632.186,A -85,B 0,C 180,E1 -4052.248,E2 -4052.248} C_VEL
LIN {X 0,Y 537.561,Z 629.882,A -85,B 0,C 180,E1 -4053.748,E2 -4053.748} C_VEL
LIN {X 0,Y 537.574,Z 626.386,A -85,B 0,C 180,E1 -4055.251,E2 -4055.251} C_VEL
LIN {X 0,Y 537.62,Z 621.609,A -85,B 0,C 180,E1 -4056.757,E2 -4056.757} C_VEL
LIN {X 0,Y 537.735,Z 615.419,A -85,B 0,C 180,E1 -4058.266,E2 -4058.266} C_VEL
LIN {X 0,Y 537.86,Z 607.642,A -85,B 0,C 180,E1 -4059.78,E2 -4059.78} C_VEL
LIN {X 0,Y 538.102,Z 599.366,A -85,B 0,C 180,E1 -4061.107,E2 -4061.107} C_VEL
LIN {X 0,Y 538.359,Z 589.391,A -85,B 0,C 180,E1 -4062.439,E2 -4062.439} C_VEL
LIN {X 0,Y 538.663,Z 579.183,A -85,B 0,C 180,E1 -4063.583,E2 -4063.583} C_VEL
LIN {X 0,Y 539.023,Z 566.953,A -85,B 0,C 180,E1 -4064.729,E2 -4064.729} C_VEL
LIN {X 0,Y 539.459,Z 554.692,A -85,B 0,C 180,E1 -4065.682,E2 -4065.682} C_VEL
LIN {X 0,Y 539.82,Z 541.297,A -85,B 0,C 180,E1 -4066.546,E2 -4066.546} C_VEL
LIN {X 0,Y 540.227,Z 526.54,A -85,B 0,C 180,E1 -4067.313,E2 -4067.313} C_VEL
LIN {X 0,Y 540.534,Z 512.258,A -85,B 0,C 180,E1 -4067.889,E2 -4067.889} C_VEL
LIN {X 0,Y 540.82,Z 497.367,A -85,B 0,C 180,E1 -4068.332,E2 -4068.332} C_VEL
LIN {X 0,Y 541.038,Z 482.333,A -85,B 0,C 180,E1 -4068.628,E2 -4068.628} C_VEL
LIN {X 0,Y 541.772,Z 332.85,A -85,B 0,C 180,E1 -4070.668,E2 -4070.668} C_VEL
LIN {X 0,Y 539.533,Z 321.346,A -85,B 0,C 180,E1 -4070.932,E2 -4070.932} C_VEL
LIN {X 0,Y 540.113,Z 298.829,A -85,B 0,C 180,E1 -4073.789,E2 -4073.789} C_VEL
LIN {X 0,Y 540.439,Z 281.752,A -85,B 0,C 180,E1 -4075.997,E2 -4075.997} C_VEL
LIN {X 0,Y 538,Z 271.092,A -85,B 0,C 180,E1 -4077.561,E2 -4077.561} C_VEL
LIN {X 0,Y 538.016,Z 271.091,A -85,B 0,C 180,E1 -4080.441,E2 -4080.441} C_VEL
LIN {X 0,Y 538.02,Z 271.089,A -85,B 0,C 180,E1 -4083.278,E2 -4083.278} C_VEL
LIN {X 0,Y 537.986,Z 271.099,A -85,B 0,C 180,E1 -4086.005,E2 -4086.005} C_VEL
LIN {X 0,Y 538.008,Z 271.091,A -85,B 0,C 180,E1 -4088.83,E2 -4088.83} C_VEL
LIN {X 0,Y 537.988,Z 271.097,A -85,B 0,C 180,E1 -4091.873,E2 -4091.873} C_VEL
LIN {X 0,Y 537.991,Z 271.091,A -85,B 0,C 180,E1 -4094.863,E2 -4094.863} C_VEL
LIN {X 0,Y 537.985,Z 271.091,A -85,B 0,C 180,E1 -4097.21,E2 -4097.21} C_VEL
LIN {X 0,Y 538.007,Z 271.09,A -85,B 0,C 180,E1 -4100.417,E2 -4100.417} C_VEL
LIN {X 0,Y 537.954,Z 271.097,A -85,B 0,C 180,E1 -4103.061,E2 -4103.061} C_VEL
LIN {X 0,Y 537.994,Z 271.095,A -85,B 0,C 180,E1 -4105.824,E2 -4105.824} C_VEL
LIN {X 0,Y 538.004,Z 271.09,A -85,B 0,C 180,E1 -4108.498,E2 -4108.498} C_VEL
LIN {X 0,Y 538.015,Z 271.088,A -85,B 0,C 180,E1 -4111.096,E2 -4111.096} C_VEL
LIN {X 0,Y 537.975,Z 271.098,A -85,B 0,C 180,E1 -4113.629,E2 -4113.629} C_VEL
LIN {X 0,Y 538.002,Z 271.094,A -85,B 0,C 180,E1 -4116.121,E2 -4116.121} C_VEL
LIN {X 0,Y 538.03,Z 271.09,A -85,B 0,C 180,E1 -4119.347,E2 -4119.347} C_VEL
LIN {X 0,Y 537.999,Z 271.099,A -85,B 0,C 180,E1 -4121.728,E2 -4121.728} C_VEL
LIN {X 0,Y 538.053,Z 271.084,A -85,B 0,C 180,E1 -4125.142,E2 -4125.142} C_VEL
LIN {X 0,Y 538.035,Z 271.081,A -85,B 0,C 180,E1 -4128.424,E2 -4128.424} C_VEL
LIN {X 0,Y 538.025,Z 271.094,A -85,B 0,C 180,E1 -4131.738,E2 -4131.738} C_VEL
LIN {X 0,Y 538.119,Z 271.072,A -85,B 0,C 180,E1 -4134.753,E2 -4134.753} C_VEL
LIN {X 0,Y 538.144,Z 271.074,A -85,B 0,C 180,E1 -4137.753,E2 -4137.753} C_VEL
LIN {X 0,Y 538.139,Z 271.074,A -85,B 0,C 180,E1 -4139.999,E2 -4139.999} C_VEL
LIN {X 0,Y 538.11,Z 271.077,A -85,B 0,C 180,E1 -4142.993,E2 -4142.993} C_VEL
LIN {X 0,Y 538.057,Z 271.075,A -85,B 0,C 180,E1 -4145.997,E2 -4145.997} C_VEL
LIN {X 0,Y 538.009,Z 271.087,A -85,B 0,C 180,E1 -4149.017,E2 -4149.017} C_VEL
LIN {X 0,Y 538.037,Z 271.086,A -85,B 0,C 180,E1 -4152.062,E2 -4152.062} C_VEL
LIN {X 0,Y 538.024,Z 271.09,A -85,B 0,C 180,E1 -4155.143,E2 -4155.143} C_VEL
LIN {X 0,Y 537.992,Z 271.085,A -85,B 0,C 180,E1 -4158.27,E2 -4158.27} C_VEL
LIN {X 0,Y 538.019,Z 271.087,A -85,B 0,C 180,E1 -4160.65,E2 -4160.65} C_VEL
LIN {X 0,Y 537.992,Z 271.09,A -85,B 0,C 180,E1 -4163.876,E2 -4163.876} C_VEL
LIN {X 0,Y 537.974,Z 271.086,A -85,B 0,C 180,E1 -4166.368,E2 -4166.368} C_VEL
LIN {X 0,Y 537.977,Z 271.091,A -85,B 0,C 180,E1 -4168.925,E2 -4168.925} C_VEL
LIN {X 0,Y 537.994,Z 271.091,A -85,B 0,C 180,E1 -4171.886,E2 -4171.886} C_VEL
LIN {X 0,Y 537.981,Z 271.092,A -85,B 0,C 180,E1 -4174.614,E2 -4174.614} C_VEL
LIN {X 0,Y 537.982,Z 271.093,A -85,B 0,C 180,E1 -4177.168,E2 -4177.168} C_VEL
LIN {X 0,Y 538.005,Z 271.089,A -85,B 0,C 180,E1 -4179.796,E2 -4179.796} C_VEL
LIN {X 0,Y 537.98,Z 271.092,A -85,B 0,C 180,E1 -4180.209,E2 -4180.209} C_VEL
LIN {X 0,Y 537.311,Z 271.182,A -85,B 0,C 180,E1 -4180.834,E2 -4180.834} C_VEL
LIN {X 0,Y 534.462,Z 271.536,A -85,B 0,C 180,E1 -4181.849,E2 -4181.849} C_VEL
LIN {X 0,Y 532.054,Z 271.836,A -85,B 0,C 180,E1 -4182.666,E2 -4182.666} C_VEL
LIN {X 0,Y 531.014,Z 271.963,A -85,B 0,C 180,E1 -4183.297,E2 -4183.297} C_VEL
LIN {X 0,Y 530.927,Z 271.97,A -85,B 0,C 180,E1 -4183.51,E2 -4183.51} C_VEL
LIN {X 0,Y 530.92,Z 271.969,A -85,B 0,C 180,E1 -4186.502,E2 -4186.502} C_VEL
LIN {X 0,Y 530.962,Z 271.968,A -85,B 0,C 180,E1 -4189.566,E2 -4189.566} C_VEL
LIN {X 0,Y 530.949,Z 271.969,A -85,B 0,C 180,E1 -4192.576,E2 -4192.576} C_VEL
LIN {X 0,Y 530.973,Z 271.969,A -85,B 0,C 180,E1 -4195.309,E2 -4195.309} C_VEL
LIN {X 0,Y 530.948,Z 271.967,A -85,B 0,C 180,E1 -4198.031,E2 -4198.031} C_VEL
LIN {X 0,Y 530.969,Z 271.971,A -85,B 0,C 180,E1 -4200.874,E2 -4200.874} C_VEL
LIN {X 0,Y 530.982,Z 271.966,A -85,B 0,C 180,E1 -4203.255,E2 -4203.255} C_VEL
LIN {X 0,Y 530.939,Z 271.968,A -85,B 0,C 180,E1 -4205.967,E2 -4205.967} C_VEL
LIN {X 0,Y 530.98,Z 271.967,A -85,B 0,C 180,E1 -4209.061,E2 -4209.061} C_VEL
LIN {X 0,Y 530.998,Z 271.965,A -85,B 0,C 180,E1 -4212.277,E2 -4212.277} C_VEL
LIN {X 0,Y 530.999,Z 271.962,A -85,B 0,C 180,E1 -4215.435,E2 -4215.435} C_VEL
LIN {X 0,Y 531.036,Z 271.965,A -85,B 0,C 180,E1 -4218.55,E2 -4218.55} C_VEL
LIN {X 0,Y 531.032,Z 271.957,A -85,B 0,C 180,E1 -4221.629,E2 -4221.629} C_VEL
LIN {X 0,Y 531.102,Z 271.958,A -85,B 0,C 180,E1 -4224.685,E2 -4224.685} C_VEL
LIN {X 0,Y 531.115,Z 271.949,A -85,B 0,C 180,E1 -4227.725,E2 -4227.725} C_VEL
LIN {X 0,Y 531.139,Z 271.954,A -85,B 0,C 180,E1 -4230.758,E2 -4230.758} C_VEL
LIN {X 0,Y 531.091,Z 271.957,A -85,B 0,C 180,E1 -4233.034,E2 -4233.034} C_VEL
LIN {X 0,Y 531.081,Z 271.975,A -85,B 0,C 180,E1 -4235.458,E2 -4235.458} C_VEL
LIN {X 0,Y 532.887,Z 281.422,A -85,B 0,C 180,E1 -4237.007,E2 -4237.007} C_VEL
LIN {X 0,Y 532.576,Z 293.803,A -85,B 0,C 180,E1 -4238.857,E2 -4238.857} C_VEL
LIN {X 0,Y 535.184,Z 305.813,A -85,B 0,C 180,E1 -4239.138,E2 -4239.138} C_VEL
LIN {X 0,Y 534.28,Z 458.019,A -85,B 0,C 180,E1 -4241.259,E2 -4241.259} C_VEL
LIN {X 0,Y 534.045,Z 473.538,A -85,B 0,C 180,E1 -4241.625,E2 -4241.625} C_VEL
LIN {X 0,Y 533.698,Z 487.961,A -85,B 0,C 180,E1 -4242.114,E2 -4242.114} C_VEL
LIN {X 0,Y 533.295,Z 503.008,A -85,B 0,C 180,E1 -4242.796,E2 -4242.796} C_VEL
LIN {X 0,Y 532.832,Z 517.522,A -85,B 0,C 180,E1 -4243.636,E2 -4243.636} C_VEL
LIN {X 0,Y 532.436,Z 529.972,A -85,B 0,C 180,E1 -4244.524,E2 -4244.524} C_VEL
LIN {X 0,Y 532.024,Z 541.387,A -85,B 0,C 180,E1 -4245.495,E2 -4245.495} C_VEL
LIN {X 0,Y 531.593,Z 553.329,A -85,B 0,C 180,E1 -4246.711,E2 -4246.711} C_VEL
LIN {X 0,Y 531.269,Z 563.064,A -85,B 0,C 180,E1 -4247.892,E2 -4247.892} C_VEL
LIN {X 0,Y 530.963,Z 572.911,A -85,B 0,C 180,E1 -4249.323,E2 -4249.323} C_VEL
LIN {X 0,Y 530.72,Z 580.983,A -85,B 0,C 180,E1 -4250.746,E2 -4250.746} C_VEL
LIN {X 0,Y 530.582,Z 587.985,A -85,B 0,C 180,E1 -4252.262,E2 -4252.262} C_VEL
LIN {X 0,Y 530.534,Z 592.395,A -85,B 0,C 180,E1 -4253.416,E2 -4253.416} C_VEL
LIN {X 0,Y 530.473,Z 597.357,A -85,B 0,C 180,E1 -4255.084,E2 -4255.084} C_VEL
LIN {X 0,Y 530.343,Z 600.85,A -85,B 0,C 180,E1 -4256.779,E2 -4256.779} C_VEL
LIN {X 0,Y 530.363,Z 602.888,A -85,B 0,C 180,E1 -4258.492,E2 -4258.492} C_VEL
LIN {X 0,Y 530.402,Z 603.468,A -85,B 0,C 180,E1 -4260.232,E2 -4260.232} C_VEL
LIN {X 0,Y 530.355,Z 602.518,A -85,B 0,C 180,E1 -4262.008,E2 -4262.008} C_VEL
LIN {X 0,Y 530.355,Z 600.71,A -85,B 0,C 180,E1 -4263.404,E2 -4263.404} C_VEL
LIN {X 0,Y 530.419,Z 596.856,A -85,B 0,C 180,E1 -4265.194,E2 -4265.194} C_VEL
LIN {X 0,Y 530.526,Z 592.674,A -85,B 0,C 180,E1 -4266.592,E2 -4266.592} C_VEL
LIN {X 0,Y 530.635,Z 586.203,A -85,B 0,C 180,E1 -4268.255,E2 -4268.255} C_VEL
LIN {X 0,Y 530.816,Z 579.424,A -85,B 0,C 180,E1 -4269.649,E2 -4269.649} C_VEL
LIN {X 0,Y 531.037,Z 571.258,A -85,B 0,C 180,E1 -4271.033,E2 -4271.033} C_VEL
LIN {X 0,Y 531.302,Z 561.384,A -85,B 0,C 180,E1 -4272.423,E2 -4272.423} C_VEL
LIN {X 0,Y 531.689,Z 550.633,A -85,B 0,C 180,E1 -4273.68,E2 -4273.68} C_VEL
LIN {X 0,Y 532.105,Z 539.054,A -85,B 0,C 180,E1 -4274.812,E2 -4274.812} C_VEL
LIN {X 0,Y 532.557,Z 525.697,A -85,B 0,C 180,E1 -4275.895,E2 -4275.895} C_VEL
LIN {X 0,Y 533.021,Z 512.296,A -85,B 0,C 180,E1 -4276.783,E2 -4276.783} C_VEL
LIN {X 0,Y 533.449,Z 498.071,A -85,B 0,C 180,E1 -4277.541,E2 -4277.541} C_VEL
LIN {X 0,Y 533.795,Z 483.288,A -85,B 0,C 180,E1 -4278.154,E2 -4278.154} C_VEL
LIN {X 0,Y 534.134,Z 468.094,A -85,B 0,C 180,E1 -4278.614,E2 -4278.614} C_VEL
LIN {X 0,Y 534.336,Z 451.997,A -85,B 0,C 180,E1 -4278.931,E2 -4278.931} C_VEL
LIN {X 0,Y 535.168,Z 305.508,A -85,B 0,C 180,E1 -4280.959,E2 -4280.959} C_VEL
LIN {X 0,Y 532.597,Z 293.689,A -85,B 0,C 180,E1 -4281.253,E2 -4281.253} C_VEL
LIN {X 0,Y 532.854,Z 281.323,A -85,B 0,C 180,E1 -4283.124,E2 -4283.124} C_VEL
LIN {X 0,Y 531.312,Z 273.54,A -85,B 0,C 180,E1 -4284.41,E2 -4284.41} C_VEL
LIN {X 0,Y 530.985,Z 271.97,A -85,B 0,C 180,E1 -4284.699,E2 -4284.699} C_VEL
LIN {X 0,Y 530.958,Z 271.974,A -85,B 0,C 180,E1 -4287.135,E2 -4287.135} C_VEL
LIN {X 0,Y 530.969,Z 271.973,A -85,B 0,C 180,E1 -4289.805,E2 -4289.805} C_VEL
LIN {X 0,Y 531.001,Z 271.963,A -85,B 0,C 180,E1 -4292.467,E2 -4292.467} C_VEL
LIN {X 0,Y 530.991,Z 271.967,A -85,B 0,C 180,E1 -4294.944,E2 -4294.944} C_VEL
LIN {X 0,Y 530.955,Z 271.968,A -85,B 0,C 180,E1 -4298.248,E2 -4298.248} C_VEL
LIN {X 0,Y 530.982,Z 271.966,A -85,B 0,C 180,E1 -4300.679,E2 -4300.679} C_VEL
LIN {X 0,Y 530.977,Z 271.973,A -85,B 0,C 180,E1 -4303.072,E2 -4303.072} C_VEL
LIN {X 0,Y 531.004,Z 271.967,A -85,B 0,C 180,E1 -4305.437,E2 -4305.437} C_VEL
LIN {X 0,Y 531.021,Z 271.961,A -85,B 0,C 180,E1 -4308.551,E2 -4308.551} C_VEL
LIN {X 0,Y 531.036,Z 271.959,A -85,B 0,C 180,E1 -4311.631,E2 -4311.631} C_VEL
LIN {X 0,Y 531.106,Z 271.952,A -85,B 0,C 180,E1 -4314.686,E2 -4314.686} C_VEL
LIN {X 0,Y 531.12,Z 271.948,A -85,B 0,C 180,E1 -4317.726,E2 -4317.726} C_VEL
LIN {X 0,Y 531.144,Z 271.951,A -85,B 0,C 180,E1 -4320.759,E2 -4320.759} C_VEL
LIN {X 0,Y 531.091,Z 271.957,A -85,B 0,C 180,E1 -4323.035,E2 -4323.035} C_VEL
LIN {X 0,Y 531.041,Z 271.957,A -85,B 0,C 180,E1 -4326.079,E2 -4326.079} C_VEL
LIN {X 0,Y 531.019,Z 271.961,A -85,B 0,C 180,E1 -4328.372,E2 -4328.372} C_VEL
LIN {X 0,Y 531.038,Z 271.956,A -85,B 0,C 180,E1 -4331.672,E2 -4331.672} C_VEL
LIN {X 0,Y 531.02,Z 271.964,A -85,B 0,C 180,E1 -4334.957,E2 -4334.957} C_VEL
LIN {X 0,Y 530.971,Z 271.965,A -85,B 0,C 180,E1 -4337.725,E2 -4337.725} C_VEL
LIN {X 0,Y 531.015,Z 271.962,A -85,B 0,C 180,E1 -4340.128,E2 -4340.128} C_VEL
LIN {X 0,Y 530.933,Z 271.977,A -85,B 0,C 180,E1 -4342.575,E2 -4342.575} C_VEL
LIN {X 0,Y 530.936,Z 271.971,A -85,B 0,C 180,E1 -4345.062,E2 -4345.062} C_VEL
LIN {X 0,Y 530.953,Z 271.968,A -85,B 0,C 180,E1 -4347.6,E2 -4347.6} C_VEL
LIN {X 0,Y 530.94,Z 271.975,A -85,B 0,C 180,E1 -4350.2,E2 -4350.2} C_VEL
LIN {X 0,Y 530.956,Z 271.969,A -85,B 0,C 180,E1 -4352.868,E2 -4352.868} C_VEL
LIN {X 0,Y 530.919,Z 271.973,A -85,B 0,C 180,E1 -4355.624,E2 -4355.624} C_VEL
LIN {X 0,Y 530.948,Z 271.97,A -85,B 0,C 180,E1 -4358.653,E2 -4358.653} C_VEL
LIN {X 0,Y 530.913,Z 271.973,A -85,B 0,C 180,E1 -4361.444,E2 -4361.444} C_VEL
LIN {X 0,Y 530.957,Z 271.971,A -85,B 0,C 180,E1 -4364.551,E2 -4364.551} C_VEL
LIN {X 0,Y 530.908,Z 271.976,A -85,B 0,C 180,E1 -4367.538,E2 -4367.538} C_VEL
LIN {X 0,Y 530.963,Z 271.969,A -85,B 0,C 180,E1 -4370.556,E2 -4370.556} C_VEL
LIN {X 0,Y 530.912,Z 271.973,A -85,B 0,C 180,E1 -4373.439,E2 -4373.439} C_VEL
LIN {X 0,Y 530.976,Z 271.968,A -85,B 0,C 180,E1 -4376.499,E2 -4376.499} C_VEL
LIN {X 0,Y 530.965,Z 271.97,A -85,B 0,C 180,E1 -4379.357,E2 -4379.357} C_VEL
LIN {X 0,Y 530.97,Z 271.989,A -85,B 0,C 180,E1 -4382.242,E2 -4382.242} C_VEL
LIN {X 0,Y 533.613,Z 283.674,A -85,B 0,C 180,E1 -4383.949,E2 -4383.949} C_VEL
LIN {X 0,Y 533.16,Z 301.646,A -85,B 0,C 180,E1 -4386.295,E2 -4386.295} C_VEL
LIN {X 0,Y 532.617,Z 321.113,A -85,B 0,C 180,E1 -4388.796,E2 -4388.796} C_VEL
LIN {X 0,Y 535.168,Z 334.92,A -85,B 0,C 180,E1 -4389.099,E2 -4389.099} C_VEL
LIN {X 0,Y 534.251,Z 487.321,A -85,B 0,C 180,E1 -4391.218,E2 -4391.218} C_VEL
LIN {X 0,Y 533.976,Z 502.914,A -85,B 0,C 180,E1 -4391.587,E2 -4391.587} C_VEL
LIN {X 0,Y 533.656,Z 517.119,A -85,B 0,C 180,E1 -4392.072,E2 -4392.072} C_VEL
LIN {X 0,Y 533.245,Z 531.216,A -85,B 0,C 180,E1 -4392.701,E2 -4392.701} C_VEL
LIN {X 0,Y 532.837,Z 544.191,A -85,B 0,C 180,E1 -4393.428,E2 -4393.428} C_VEL
LIN {X 0,Y 532.452,Z 556.992,A -85,B 0,C 180,E1 -4394.302,E2 -4394.302} C_VEL
LIN {X 0,Y 532,Z 569.92,A -85,B 0,C 180,E1 -4395.366,E2 -4395.366} C_VEL
LIN {X 0,Y 531.621,Z 580.747,A -85,B 0,C 180,E1 -4396.429,E2 -4396.429} C_VEL
LIN {X 0,Y 531.293,Z 590.762,A -85,B 0,C 180,E1 -4397.588,E2 -4397.588} C_VEL
LIN {X 0,Y 531.062,Z 600.559,A -85,B 0,C 180,E1 -4398.937,E2 -4398.937} C_VEL
LIN {X 0,Y 530.78,Z 608.726,A -85,B 0,C 180,E1 -4400.281,E2 -4400.281} C_VEL
LIN {X 0,Y 530.665,Z 615.425,A -85,B 0,C 180,E1 -4401.624,E2 -4401.624} C_VEL
LIN {X 0,Y 530.55,Z 621.607,A -85,B 0,C 180,E1 -4403.153,E2 -4403.153} C_VEL
LIN {X 0,Y 530.508,Z 626.387,A -85,B 0,C 180,E1 -4404.68,E2 -4404.68} C_VEL
LIN {X 0,Y 530.48,Z 629.887,A -85,B 0,C 180,E1 -4406.202,E2 -4406.202} C_VEL
LIN {X 0,Y 530.408,Z 632.189,A -85,B 0,C 180,E1 -4407.722,E2 -4407.722} C_VEL
LIN {X 0,Y 530.342,Z 633.347,A -85,B 0,C 180,E1 -4409.241,E2 -4409.241} C_VEL
LIN {X 0,Y 530.342,Z 633.346,A -85,B 0,C 180,E1 -4410.76,E2 -4410.76} C_VEL
LIN {X 0,Y 530.409,Z 632.185,A -85,B 0,C 180,E1 -4412.278,E2 -4412.278} C_VEL
LIN {X 0,Y 530.48,Z 629.881,A -85,B 0,C 180,E1 -4413.798,E2 -4413.798} C_VEL
LIN {X 0,Y 530.508,Z 626.386,A -85,B 0,C 180,E1 -4415.321,E2 -4415.321} C_VEL
LIN {X 0,Y 530.551,Z 621.609,A -85,B 0,C 180,E1 -4416.847,E2 -4416.847} C_VEL
LIN {X 0,Y 530.666,Z 615.419,A -85,B 0,C 180,E1 -4418.377,E2 -4418.377} C_VEL
LIN {X 0,Y 530.809,Z 607.63,A -85,B 0,C 180,E1 -4419.911,E2 -4419.911} C_VEL
LIN {X 0,Y 531.057,Z 599.292,A -85,B 0,C 180,E1 -4421.257,E2 -4421.257} C_VEL
LIN {X 0,Y 531.348,Z 589.244,A -85,B 0,C 180,E1 -4422.606,E2 -4422.606} C_VEL
LIN {X 0,Y 531.684,Z 578.966,A -85,B 0,C 180,E1 -4423.764,E2 -4423.764} C_VEL
LIN {X 0,Y 532.104,Z 566.72,A -85,B 0,C 180,E1 -4424.925,E2 -4424.925} C_VEL
LIN {X 0,Y 532.56,Z 553.218,A -85,B 0,C 180,E1 -4425.981,E2 -4425.981} C_VEL
LIN {X 0,Y 533.052,Z 539.408,A -85,B 0,C 180,E1 -4426.861,E2 -4426.861} C_VEL
LIN {X 0,Y 533.455,Z 525.24,A -85,B 0,C 180,E1 -4427.589,E2 -4427.589} C_VEL
LIN {X 0,Y 533.827,Z 509.909,A -85,B 0,C 180,E1 -4428.196,E2 -4428.196} C_VEL
LIN {X 0,Y 534.106,Z 495.032,A -85,B 0,C 180,E1 -4428.624,E2 -4428.624} C_VEL
LIN {X 0,Y 534.296,Z 478.448,A -85,B 0,C 180,E1 -4428.925,E2 -4428.925} C_VEL
LIN {X 0,Y 535.131,Z 333.917,A -85,B 0,C 180,E1 -4430.918,E2 -4430.918} C_VEL
LIN {X 0,Y 532.645,Z 321.218,A -85,B 0,C 180,E1 -4431.207,E2 -4431.207} C_VEL
LIN {X 0,Y 533.256,Z 300.231,A -85,B 0,C 180,E1 -4433.908,E2 -4433.908} C_VEL
LIN {X 0,Y 533.636,Z 283.82,A -85,B 0,C 180,E1 -4436.057,E2 -4436.057} C_VEL
LIN {X 0,Y 530.979,Z 271.965,A -85,B 0,C 180,E1 -4437.819,E2 -4437.819} C_VEL
LIN {X 0,Y 530.968,Z 271.97,A -85,B 0,C 180,E1 -4440.643,E2 -4440.643} C_VEL
LIN {X 0,Y 530.961,Z 271.97,A -85,B 0,C 180,E1 -4443.499,E2 -4443.499} C_VEL
LIN {X 0,Y 530.934,Z 271.976,A -85,B 0,C 180,E1 -4446.56,E2 -4446.56} C_VEL
LIN {X 0,Y 530.967,Z 271.969,A -85,B 0,C 180,E1 -4449.444,E2 -4449.444} C_VEL
LIN {X 0,Y 530.917,Z 271.974,A -85,B 0,C 180,E1 -4452.462,E2 -4452.462} C_VEL
LIN {X 0,Y 530.964,Z 271.968,A -85,B 0,C 180,E1 -4455.45,E2 -4455.45} C_VEL
LIN {X 0,Y 530.961,Z 271.97,A -85,B 0,C 180,E1 -4458.561,E2 -4458.561} C_VEL
LIN {X 0,Y 530.947,Z 271.97,A -85,B 0,C 180,E1 -4461.528,E2 -4461.528} C_VEL
LIN {X 0,Y 530.926,Z 271.972,A -85,B 0,C 180,E1 -4464.377,E2 -4464.377} C_VEL
LIN {X 0,Y 530.963,Z 271.966,A -85,B 0,C 180,E1 -4467.132,E2 -4467.132} C_VEL
LIN {X 0,Y 530.949,Z 271.975,A -85,B 0,C 180,E1 -4469.801,E2 -4469.801} C_VEL
LIN {X 0,Y 530.958,Z 271.967,A -85,B 0,C 180,E1 -4472.477,E2 -4472.477} C_VEL
LIN {X 0,Y 530.941,Z 271.97,A -85,B 0,C 180,E1 -4474.938,E2 -4474.938} C_VEL
LIN {X 0,Y 530.973,Z 271.974,A -85,B 0,C 180,E1 -4477.897,E2 -4477.897} C_VEL
LIN {X 0,Y 530.974,Z 271.964,A -85,B 0,C 180,E1 -4480.676,E2 -4480.676} C_VEL
LIN {X 0,Y 530.947,Z 271.97,A -85,B 0,C 180,E1 -4483.069,E2 -4483.069} C_VEL
LIN {X 0,Y 531.011,Z 271.964,A -85,B 0,C 180,E1 -4485.435,E2 -4485.435} C_VEL
LIN {X 0,Y 530.982,Z 271.958,A -85,B 0,C 180,E1 -4488.547,E2 -4488.547} C_VEL
LIN {X 0,Y 530.974,Z 271.973,A -85,B 0,C 180,E1 -4491.627,E2 -4491.627} C_VEL
LIN {X 0,Y 531.079,Z 271.949,A -85,B 0,C 180,E1 -4494.684,E2 -4494.684} C_VEL
LIN {X 0,Y 531.117,Z 271.949,A -85,B 0,C 180,E1 -4497.724,E2 -4497.724} C_VEL
LIN {X 0,Y 531.108,Z 271.95,A -85,B 0,C 180,E1 -4499.999,E2 -4499.999} C_VEL
LIN {X 0,Y 531.078,Z 271.954,A -85,B 0,C 180,E1 -4503.033,E2 -4503.033} C_VEL
LIN {X 0,Y 531.015,Z 271.951,A -85,B 0,C 180,E1 -4506.077,E2 -4506.077} C_VEL
LIN {X 0,Y 530.976,Z 271.965,A -85,B 0,C 180,E1 -4509.138,E2 -4509.138} C_VEL
LIN {X 0,Y 531.035,Z 271.962,A -85,B 0,C 180,E1 -4511.667,E2 -4511.667} C_VEL
LIN {X 0,Y 531.006,Z 271.961,A -85,B 0,C 180,E1 -4514.949,E2 -4514.949} C_VEL
LIN {X 0,Y 530.959,Z 271.964,A -85,B 0,C 180,E1 -4517.723,E2 -4517.723} C_VEL
LIN {X 0,Y 531.001,Z 271.96,A -85,B 0,C 180,E1 -4520.126,E2 -4520.126} C_VEL
LIN {X 0,Y 530.926,Z 271.971,A -85,B 0,C 180,E1 -4522.572,E2 -4522.572} C_VEL
LIN {X 0,Y 530.938,Z 271.973,A -85,B 0,C 180,E1 -4525.059,E2 -4525.059} C_VEL
LIN {X 0,Y 530.944,Z 271.966,A -85,B 0,C 180,E1 -4527.597,E2 -4527.597} C_VEL
LIN {X 0,Y 530.944,Z 271.969,A -85,B 0,C 180,E1 -4530.641,E2 -4530.641} C_VEL
LIN {X 0,Y 530.945,Z 271.971,A -85,B 0,C 180,E1 -4533.498,E2 -4533.498} C_VEL
LIN {X 0,Y 530.933,Z 271.964,A -85,B 0,C 180,E1 -4536.558,E2 -4536.558} C_VEL
LIN {X 0,Y 530.969,Z 271.969,A -85,B 0,C 180,E1 -4539.442,E2 -4539.442} C_VEL
LIN {X 0,Y 530.921,Z 271.973,A -85,B 0,C 180,E1 -4542.46,E2 -4542.46} C_VEL
LIN {X 0,Y 530.927,Z 271.97,A -85,B 0,C 180,E1 -4543.51,E2 -4543.51} C_VEL
LIN {X 0,Y 530.253,Z 272.051,A -85,B 0,C 180,E1 -4544.144,E2 -4544.144} C_VEL
LIN {X 0,Y 527.399,Z 272.411,A -85,B 0,C 180,E1 -4545.173,E2 -4545.173} C_VEL
LIN {X 0,Y 524.991,Z 272.713,A -85,B 0,C 180,E1 -4546.001,E2 -4546.001} C_VEL
LIN {X 0,Y 523.958,Z 272.84,A -85,B 0,C 180,E1 -4546.641,E2 -4546.641} C_VEL
LIN {X 0,Y 523.874,Z 272.85,A -85,B 0,C 180,E1 -4546.857,E2 -4546.857} C_VEL
LIN {X 0,Y 523.919,Z 272.851,A -85,B 0,C 180,E1 -4548.906,E2 -4548.906} C_VEL
LIN {X 0,Y 523.896,Z 272.844,A -85,B 0,C 180,E1 -4551.897,E2 -4551.897} C_VEL
LIN {X 0,Y 523.911,Z 272.851,A -85,B 0,C 180,E1 -4554.91,E2 -4554.91} C_VEL
LIN {X 0,Y 523.916,Z 272.844,A -85,B 0,C 180,E1 -4557.679,E2 -4557.679} C_VEL
LIN {X 0,Y 523.934,Z 272.844,A -85,B 0,C 180,E1 -4560.676,E2 -4560.676} C_VEL
LIN {X 0,Y 523.954,Z 272.838,A -85,B 0,C 180,E1 -4563.728,E2 -4563.728} C_VEL
LIN {X 0,Y 523.893,Z 272.848,A -85,B 0,C 180,E1 -4566.269,E2 -4566.269} C_VEL
LIN {X 0,Y 523.927,Z 272.849,A -85,B 0,C 180,E1 -4568.766,E2 -4568.766} C_VEL
LIN {X 0,Y 523.932,Z 272.846,A -85,B 0,C 180,E1 -4571.22,E2 -4571.22} C_VEL
LIN {X 0,Y 523.916,Z 272.842,A -85,B 0,C 180,E1 -4573.638,E2 -4573.638} C_VEL
LIN {X 0,Y 523.919,Z 272.845,A -85,B 0,C 180,E1 -4576.027,E2 -4576.027} C_VEL
LIN {X 0,Y 523.995,Z 272.835,A -85,B 0,C 180,E1 -4579.177,E2 -4579.177} C_VEL
LIN {X 0,Y 524.008,Z 272.837,A -85,B 0,C 180,E1 -4582.292,E2 -4582.292} C_VEL
LIN {X 0,Y 524.062,Z 272.834,A -85,B 0,C 180,E1 -4584.613,E2 -4584.613} C_VEL
LIN {X 0,Y 524.088,Z 272.825,A -85,B 0,C 180,E1 -4587.694,E2 -4587.694} C_VEL
LIN {X 0,Y 524.108,Z 272.83,A -85,B 0,C 180,E1 -4590.768,E2 -4590.768} C_VEL
LIN {X 0,Y 524.056,Z 272.834,A -85,B 0,C 180,E1 -4593.075,E2 -4593.075} C_VEL
LIN {X 0,Y 524.064,Z 272.985,A -85,B 0,C 180,E1 -4595.241,E2 -4595.241} C_VEL
LIN {X 0,Y 526.037,Z 282.997,A -85,B 0,C 180,E1 -4596.906,E2 -4596.906} C_VEL
LIN {X 0,Y 525.748,Z 293.751,A -85,B 0,C 180,E1 -4598.552,E2 -4598.552} C_VEL
LIN {X 0,Y 528.496,Z 306.556,A -85,B 0,C 180,E1 -4598.868,E2 -4598.868} C_VEL
LIN {X 0,Y 527.693,Z 438.604,A -85,B 0,C 180,E1 -4600.722,E2 -4600.722} C_VEL
LIN {X 0,Y 527.524,Z 460.89,A -85,B 0,C 180,E1 -4601.065,E2 -4601.065} C_VEL
LIN {X 0,Y 527.248,Z 476.307,A -85,B 0,C 180,E1 -4601.46,E2 -4601.46} C_VEL
LIN {X 0,Y 526.877,Z 490.652,A -85,B 0,C 180,E1 -4601.98,E2 -4601.98} C_VEL
LIN {X 0,Y 526.451,Z 504.734,A -85,B 0,C 180,E1 -4602.649,E2 -4602.649} C_VEL
LIN {X 0,Y 525.959,Z 519.284,A -85,B 0,C 180,E1 -4603.523,E2 -4603.523} C_VEL
LIN {X 0,Y 525.476,Z 532.723,A -85,B 0,C 180,E1 -4604.523,E2 -4604.523} C_VEL
LIN {X 0,Y 524.969,Z 545.005,A -85,B 0,C 180,E1 -4605.629,E2 -4605.629} C_VEL
LIN {X 0,Y 524.562,Z 555.361,A -85,B 0,C 180,E1 -4606.741,E2 -4606.741} C_VEL
LIN {X 0,Y 524.243,Z 564.946,A -85,B 0,C 180,E1 -4607.958,E2 -4607.958} C_VEL
LIN {X 0,Y 523.948,Z 573.139,A -85,B 0,C 180,E1 -4609.185,E2 -4609.185} C_VEL
LIN {X 0,Y 523.69,Z 581.203,A -85,B 0,C 180,E1 -4610.626,E2 -4610.626} C_VEL
LIN {X 0,Y 523.513,Z 588.115,A -85,B 0,C 180,E1 -4612.14,E2 -4612.14} C_VEL
LIN {X 0,Y 523.422,Z 593.922,A -85,B 0,C 180,E1 -4613.753,E2 -4613.753} C_VEL
LIN {X 0,Y 523.376,Z 598.464,A -85,B 0,C 180,E1 -4615.448,E2 -4615.448} C_VEL
LIN {X 0,Y 523.264,Z 601.574,A -85,B 0,C 180,E1 -4617.171,E2 -4617.171} C_VEL
LIN {X 0,Y 523.264,Z 603.244,A -85,B 0,C 180,E1 -4618.914,E2 -4618.914} C_VEL
LIN {X 0,Y 523.291,Z 603.536,A -85,B 0,C 180,E1 -4619.796,E2 -4619.796} C_VEL
LIN {X 0,Y 523.282,Z 603.447,A -85,B 0,C 180,E1 -4620.737,E2 -4620.737} C_VEL
LIN {X 0,Y 523.245,Z 602.143,A -85,B 0,C 180,E1 -4622.496,E2 -4622.496} C_VEL
LIN {X 0,Y 523.278,Z 600.496,A -85,B 0,C 180,E1 -4623.626,E2 -4623.626} C_VEL
LIN {X 0,Y 523.329,Z 596.978,A -85,B 0,C 180,E1 -4625.271,E2 -4625.271} C_VEL
LIN {X 0,Y 523.453,Z 592.718,A -85,B 0,C 180,E1 -4626.72,E2 -4626.72} C_VEL
LIN {X 0,Y 523.56,Z 587.39,A -85,B 0,C 180,E1 -4628.131,E2 -4628.131} C_VEL
LIN {X 0,Y 523.738,Z 580.553,A -85,B 0,C 180,E1 -4629.597,E2 -4629.597} C_VEL
LIN {X 0,Y 523.996,Z 572.053,A -85,B 0,C 180,E1 -4631.085,E2 -4631.085} C_VEL
LIN {X 0,Y 524.29,Z 562.22,A -85,B 0,C 180,E1 -4632.504,E2 -4632.504} C_VEL
LIN {X 0,Y 524.717,Z 552.481,A -85,B 0,C 180,E1 -4633.678,E2 -4633.678} C_VEL
LIN {X 0,Y 525.134,Z 541.235,A -85,B 0,C 180,E1 -4634.824,E2 -4634.824} C_VEL
LIN {X 0,Y 525.605,Z 528.958,A -85,B 0,C 180,E1 -4635.87,E2 -4635.87} C_VEL
LIN {X 0,Y 526.113,Z 514.875,A -85,B 0,C 180,E1 -4636.855,E2 -4636.855} C_VEL
LIN {X 0,Y 526.572,Z 500.709,A -85,B 0,C 180,E1 -4637.651,E2 -4637.651} C_VEL
LIN {X 0,Y 527.006,Z 485.567,A -85,B 0,C 180,E1 -4638.312,E2 -4638.312} C_VEL
LIN {X 0,Y 527.391,Z 470.165,A -85,B 0,C 180,E1 -4638.806,E2 -4638.806} C_VEL
LIN {X 0,Y 527.601,Z 455.103,A -85,B 0,C 180,E1 -4639.13,E2 -4639.13} C_VEL
LIN {X 0,Y 528.571,Z 307.06,A -85,B 0,C 180,E1 -4641.213,E2 -4641.213} C_VEL
LIN {X 0,Y 525.74,Z 293.871,A -85,B 0,C 180,E1 -4641.551,E2 -4641.551} C_VEL
LIN {X 0,Y 525.954,Z 282.522,A -85,B 0,C 180,E1 -4643.295,E2 -4643.295} C_VEL
LIN {X 0,Y 523.936,Z 272.849,A -85,B 0,C 180,E1 -4644.936,E2 -4644.936} C_VEL
LIN {X 0,Y 523.926,Z 272.851,A -85,B 0,C 180,E1 -4647.679,E2 -4647.679} C_VEL
LIN {X 0,Y 523.952,Z 272.843,A -85,B 0,C 180,E1 -4650.674,E2 -4650.674} C_VEL
LIN {X 0,Y 523.961,Z 272.845,A -85,B 0,C 180,E1 -4653.73,E2 -4653.73} C_VEL
LIN {X 0,Y 523.92,Z 272.846,A -85,B 0,C 180,E1 -4656.272,E2 -4656.272} C_VEL
LIN {X 0,Y 523.931,Z 272.845,A -85,B 0,C 180,E1 -4658.768,E2 -4658.768} C_VEL
LIN {X 0,Y 523.939,Z 272.847,A -85,B 0,C 180,E1 -4661.222,E2 -4661.222} C_VEL
LIN {X 0,Y 523.925,Z 272.848,A -85,B 0,C 180,E1 -4663.64,E2 -4663.64} C_VEL
LIN {X 0,Y 523.925,Z 272.844,A -85,B 0,C 180,E1 -4666.029,E2 -4666.029} C_VEL
LIN {X 0,Y 523.997,Z 272.835,A -85,B 0,C 180,E1 -4668.395,E2 -4668.395} C_VEL
LIN {X 0,Y 523.985,Z 272.839,A -85,B 0,C 180,E1 -4671.517,E2 -4671.517} C_VEL
LIN {X 0,Y 524.067,Z 272.828,A -85,B 0,C 180,E1 -4674.615,E2 -4674.615} C_VEL
LIN {X 0,Y 524.093,Z 272.823,A -85,B 0,C 180,E1 -4677.696,E2 -4677.696} C_VEL
LIN {X 0,Y 524.113,Z 272.826,A -85,B 0,C 180,E1 -4680.77,E2 -4680.77} C_VEL
LIN {X 0,Y 524.056,Z 272.833,A -85,B 0,C 180,E1 -4683.076,E2 -4683.076} C_VEL
LIN {X 0,Y 524.006,Z 272.834,A -85,B 0,C 180,E1 -4686.161,E2 -4686.161} C_VEL
LIN {X 0,Y 523.973,Z 272.84,A -85,B 0,C 180,E1 -4689.263,E2 -4689.263} C_VEL
LIN {X 0,Y 523.988,Z 272.835,A -85,B 0,C 180,E1 -4691.738,E2 -4691.738} C_VEL
LIN {X 0,Y 523.983,Z 272.84,A -85,B 0,C 180,E1 -4695.053,E2 -4695.053} C_VEL
LIN {X 0,Y 523.937,Z 272.842,A -85,B 0,C 180,E1 -4697.971,E2 -4697.971} C_VEL
LIN {X 0,Y 523.962,Z 272.844,A -85,B 0,C 180,E1 -4700.411,E2 -4700.411} C_VEL
LIN {X 0,Y 523.898,Z 272.849,A -85,B 0,C 180,E1 -4702.895,E2 -4702.895} C_VEL
LIN {X 0,Y 523.886,Z 272.847,A -85,B 0,C 180,E1 -4705.423,E2 -4705.423} C_VEL
LIN {X 0,Y 523.904,Z 272.849,A -85,B 0,C 180,E1 -4708.004,E2 -4708.004} C_VEL
LIN {X 0,Y 523.906,Z 272.849,A -85,B 0,C 180,E1 -4710.648,E2 -4710.648} C_VEL
LIN {X 0,Y 523.918,Z 272.845,A -85,B 0,C 180,E1 -4713.73,E2 -4713.73} C_VEL
LIN {X 0,Y 523.852,Z 272.858,A -85,B 0,C 180,E1 -4716.396,E2 -4716.396} C_VEL
LIN {X 0,Y 523.896,Z 272.845,A -85,B 0,C 180,E1 -4719.088,E2 -4719.088} C_VEL
LIN {X 0,Y 523.886,Z 272.855,A -85,B 0,C 180,E1 -4722.126,E2 -4722.126} C_VEL
LIN {X 0,Y 523.928,Z 272.844,A -85,B 0,C 180,E1 -4725.313,E2 -4725.313} C_VEL
LIN {X 0,Y 523.911,Z 272.847,A -85,B 0,C 180,E1 -4728.696,E2 -4728.696} C_VEL
LIN {X 0,Y 523.897,Z 272.856,A -85,B 0,C 180,E1 -4731.898,E2 -4731.898} C_VEL
LIN {X 0,Y 523.912,Z 272.846,A -85,B 0,C 180,E1 -4734.914,E2 -4734.914} C_VEL
LIN {X 0,Y 523.932,Z 272.85,A -85,B 0,C 180,E1 -4737.681,E2 -4737.681} C_VEL
LIN {X 0,Y 523.951,Z 272.845,A -85,B 0,C 180,E1 -4740.678,E2 -4740.678} C_VEL
LIN {X 0,Y 523.967,Z 272.968,A -85,B 0,C 180,E1 -4742.002,E2 -4742.002} C_VEL
LIN {X 0,Y 526.821,Z 285.659,A -85,B 0,C 180,E1 -4743.882,E2 -4743.882} C_VEL
LIN {X 0,Y 526.191,Z 306.301,A -85,B 0,C 180,E1 -4746.609,E2 -4746.609} C_VEL
LIN {X 0,Y 525.738,Z 320.865,A -85,B 0,C 180,E1 -4748.503,E2 -4748.503} C_VEL
LIN {X 0,Y 528.523,Z 335.185,A -85,B 0,C 180,E1 -4748.831,E2 -4748.831} C_VEL
LIN {X 0,Y 527.52,Z 487.797,A -85,B 0,C 180,E1 -4750.987,E2 -4750.987} C_VEL
LIN {X 0,Y 527.214,Z 503.376,A -85,B 0,C 180,E1 -4751.367,E2 -4751.367} C_VEL
LIN {X 0,Y 526.84,Z 518.07,A -85,B 0,C 180,E1 -4751.882,E2 -4751.882} C_VEL
LIN {X 0,Y 526.385,Z 531.919,A -85,B 0,C 180,E1 -4752.519,E2 -4752.519} C_VEL
LIN {X 0,Y 525.919,Z 545.502,A -85,B 0,C 180,E1 -4753.304,E2 -4753.304} C_VEL
LIN {X 0,Y 525.482,Z 558.934,A -85,B 0,C 180,E1 -4754.257,E2 -4754.257} C_VEL
LIN {X 0,Y 524.953,Z 571.817,A -85,B 0,C 180,E1 -4755.364,E2 -4755.364} C_VEL
LIN {X 0,Y 524.53,Z 584.074,A -85,B 0,C 180,E1 -4756.637,E2 -4756.637} C_VEL
LIN {X 0,Y 524.138,Z 594.968,A -85,B 0,C 180,E1 -4758.005,E2 -4758.005} C_VEL
LIN {X 0,Y 523.927,Z 604.035,A -85,B 0,C 180,E1 -4759.372,E2 -4759.372} C_VEL
LIN {X 0,Y 523.678,Z 611.551,A -85,B 0,C 180,E1 -4760.733,E2 -4760.733} C_VEL
LIN {X 0,Y 523.516,Z 618.565,A -85,B 0,C 180,E1 -4762.285,E2 -4762.285} C_VEL
LIN {X 0,Y 523.431,Z 624.079,A -85,B 0,C 180,E1 -4763.834,E2 -4763.834} C_VEL
LIN {X 0,Y 523.323,Z 628.244,A -85,B 0,C 180,E1 -4765.379,E2 -4765.379} C_VEL
LIN {X 0,Y 523.359,Z 631.166,A -85,B 0,C 180,E1 -4766.921,E2 -4766.921} C_VEL
LIN {X 0,Y 523.272,Z 632.904,A -85,B 0,C 180,E1 -4768.461,E2 -4768.461} C_VEL
LIN {X 0,Y 523.244,Z 633.498,A -85,B 0,C 180,E1 -4770,E2 -4770} C_VEL
LIN {X 0,Y 523.272,Z 632.901,A -85,B 0,C 180,E1 -4771.54,E2 -4771.54} C_VEL
LIN {X 0,Y 523.359,Z 631.16,A -85,B 0,C 180,E1 -4773.079,E2 -4773.079} C_VEL
LIN {X 0,Y 523.323,Z 628.241,A -85,B 0,C 180,E1 -4774.622,E2 -4774.622} C_VEL
LIN {X 0,Y 523.431,Z 624.084,A -85,B 0,C 180,E1 -4776.166,E2 -4776.166} C_VEL
LIN {X 0,Y 523.517,Z 618.57,A -85,B 0,C 180,E1 -4777.715,E2 -4777.715} C_VEL
LIN {X 0,Y 523.7,Z 611.553,A -85,B 0,C 180,E1 -4779.267,E2 -4779.267} C_VEL
LIN {X 0,Y 523.926,Z 604.043,A -85,B 0,C 180,E1 -4780.629,E2 -4780.629} C_VEL
LIN {X 0,Y 524.151,Z 594.949,A -85,B 0,C 180,E1 -4782.001,E2 -4782.001} C_VEL
